(*appel des fonction de regulation de gaz*)
REGULATION_GAZ_L1(
	RESET:= MACHINE.STATE_Off,
	MANUAL:= MACHINE.STATE_Manu,
	VAC:= PRG_POMPAGE.VAC,
	DOOR := PRG_POMPAGE.DOOR,
	USER:= TRUE,
	PRM_Pos_Vanne:= ,
	PRM_Pressure:= ,
	PRM_Pressure_H:= ,
	PRM_Pressure_L:= ,
	PRM_Tim_Stab:= ,
 	PRM_Tim_Max_Stab:= REGULATION_GAZ_L1.PRM_Tim_Stab + T#30s,
	I_Pompage_Proc_Ok:= PRG_POMPAGE.POMPAGE.OP_Pompage_Proc.OK,
	I_Pompage_Sec_Ok:= PRG_POMPAGE.POMPAGE.OP_Pompage_Sec.EC
						OR PRG_POMPAGE.POMPAGE.OP_Pompage_Sec.OK, 	(*on n'attend pas la fin du pompage secondaire pour ne pas bloquer l'init*)
	I_Act_Pressure:= PRG_POMPAGE.M11.STATE_Pression,
	I_Marche_Gaz_Ok:= LIGNE_GAZ[1].OP_MARCHE.OK,
	I_Arret_Gaz_Ok:= LIGNE_GAZ[1].OP_ARRET.OK,
	I_Atm:= PRG_POMPAGE.POMPAGE.TH_Atm,
	PRM_Tim_Def_Pr:= (*config machine*),
	PRM_Tim_Ala_Pr:= (*config machine*),
	CONF_Flow_Init:= (*config machine*),
);

REGULATION_GAZ_L2(
	RESET:= MACHINE.STATE_Off,
	MANUAL:= MACHINE.STATE_Manu,
	VAC:= PRG_POMPAGE.VAC,
	DOOR := PRG_POMPAGE.DOOR,
	USER:= TRUE,
	PRM_Pos_Vanne:= ,
	PRM_Pressure:= ,
	PRM_Pressure_H:= ,
	PRM_Pressure_L:= ,
	PRM_Tim_Stab:= ,
 	PRM_Tim_Max_Stab:= REGULATION_GAZ_L2.PRM_Tim_Stab + T#30s,
	I_Pompage_Proc_Ok:= PRG_POMPAGE.POMPAGE.OP_Pompage_Proc.OK,
	I_Pompage_Sec_Ok:= PRG_POMPAGE.POMPAGE.OP_Pompage_Sec.EC
						OR PRG_POMPAGE.POMPAGE.OP_Pompage_Sec.OK, 	(*on n'attend pas la fin du pompage secondaire pour ne pas bloquer l'init*)
	I_Act_Pressure:= PRG_POMPAGE.M11.STATE_Pression,
	I_Marche_Gaz_Ok:= LIGNE_GAZ[2].OP_MARCHE.OK,
	I_Arret_Gaz_Ok:= LIGNE_GAZ[2].OP_ARRET.OK,
	I_Atm:= PRG_POMPAGE.POMPAGE.TH_Atm,
	PRM_Tim_Def_Pr:= (*config machine*),
	PRM_Tim_Ala_Pr:= (*config machine*),
	CONF_Flow_Init:= (*config machine*),
);

(*Affection des sorties*)
OUT_VG11	:=	LIGNE_GAZ[1].VGI.OUT_On;
OUT_VG12	:=	LIGNE_GAZ[2].VGI.OUT_On;
OUT_VG13	:=	LIGNE_GAZ[3].VGI.OUT_On;
OUT_VG14	:=	LIGNE_GAZ[4].VGI.OUT_On;
OUT_VGIN1	:=	VGIN[1].OUT_On;
OUT_VGIN2	:=	VGIN[2].OUT_On;
OUT_VGIN3	:=	VGIN[3].OUT_On;
OUT_VGIN4	:=	VGIN[4].OUT_On;

(*Affectation des état*)
STATE_AR :=((MACHINE.STATE_Auto OR MACHINE.STATE_Prod) AND LIGNE_GAZ[1].OP_ARRET.OK AND REGULATION_GAZ_L1.OP_ARRET.OK
			AND LIGNE_GAZ[2].OP_ARRET.OK AND REGULATION_GAZ_L2.OP_ARRET.OK AND
			LIGNE_GAZ[3].OP_ARRET.OK AND LIGNE_GAZ[4].OP_ARRET.OK) OR
			(MACHINE.STATE_Manu AND LIGNE_GAZ[1].VGI.STATE_Off AND LIGNE_GAZ[2].VGI.STATE_Off AND
			LIGNE_GAZ[3].VGI.STATE_Off AND LIGNE_GAZ[4].VGI.STATE_Off);

(*défaut entrainant l'arrêt du procédé*)
STATE_Def_IProc		:=		LIGNE_GAZ[1].VGI.DEF_Off_auto.DEF OR LIGNE_GAZ[1].VGI.DEF_On_Imposs.DEF OR LIGNE_GAZ[1].VGI.DEF_Off_Imposs.DEF OR
							LIGNE_GAZ[1].OP_MARCHE.DEF_ON_REJECTED.DEF OR LIGNE_GAZ[1].OP_ARRET.DEF_AUTO_ON.DEF OR
							LIGNE_GAZ[2].VGI.DEF_Off_auto.DEF OR LIGNE_GAZ[2].VGI.DEF_On_Imposs.DEF OR LIGNE_GAZ[2].VGI.DEF_Off_Imposs.DEF OR
							LIGNE_GAZ[2].OP_MARCHE.DEF_ON_REJECTED.DEF OR LIGNE_GAZ[2].OP_ARRET.DEF_AUTO_ON.DEF OR
							LIGNE_GAZ[3].VGI.DEF_Off_auto.DEF OR LIGNE_GAZ[3].VGI.DEF_On_Imposs.DEF OR LIGNE_GAZ[3].VGI.DEF_Off_Imposs.DEF OR
							LIGNE_GAZ[3].OP_MARCHE.DEF_ON_REJECTED.DEF OR LIGNE_GAZ[3].OP_ARRET.DEF_AUTO_ON.DEF OR
							LIGNE_GAZ[4].VGI.DEF_Off_auto.DEF OR LIGNE_GAZ[4].VGI.DEF_On_Imposs.DEF OR LIGNE_GAZ[4].VGI.DEF_Off_Imposs.DEF OR
							LIGNE_GAZ[4].OP_MARCHE.DEF_ON_REJECTED.DEF OR LIGNE_GAZ[4].OP_ARRET.DEF_AUTO_ON.DEF OR
							VGIN[1].DEF_Off_auto.DEF OR VGIN[1].DEF_Off_Imposs.DEF OR VGIN[1].DEF_On_Imposs.DEF OR
							VGIN[2].DEF_Off_auto.DEF OR VGIN[2].DEF_Off_Imposs.DEF OR VGIN[2].DEF_On_Imposs.DEF OR
							VGIN[3].DEF_Off_auto.DEF OR VGIN[3].DEF_Off_Imposs.DEF OR VGIN[3].DEF_On_Imposs.DEF OR
							VGIN[4].DEF_Off_auto.DEF OR VGIN[4].DEF_Off_Imposs.DEF OR VGIN[4].DEF_On_Imposs.DEF OR
							DG[1].DEF_SURV.DEF OR DG[2].DEF_SURV.DEF OR DG[3].DEF_SURV.DEF OR DG[4].DEF_SURV.DEF OR
							REGULATION_GAZ_L1.OP_MARCHE.DEF_ON_REJECTED.DEF OR REGULATION_GAZ_L1.OP_ARRET.DEF_AUTO_ON.DEF OR
							REGULATION_GAZ_L2.OP_MARCHE.DEF_ON_REJECTED.DEF OR REGULATION_GAZ_L2.OP_ARRET.DEF_AUTO_ON.DEF OR
							REGULATION_GAZ_L1.STATE_NOK OR REGULATION_GAZ_L2.STATE_NOK;

END_FUNCTION_BLOCK

// ---- POUs/Fonction/FONCTIONS GAZ/BLOCK_LIGNE_GAZ.TcPOU
FUNCTION_BLOCK BLOCK_LIGNE_GAZ
(* Gestion d'une ligne de gaz avec une vanne et un debitmètre *)

(****************historique des versions*****************************)

(* Version 1-0 - AB - VERSION INITIALE - base 6619, changement de classe de DG (MFC_BKH => MFC_MKS1179_AB*)
(* Version 2-0 - HG - Adaptation pour journal des évènements externe - 27/06/2011*)
(* Version 3.0 - AB - Variable IN_OUT DG_Prm_Flow dissociée en deux variabes, permettant de l'écrire hors appel à la fonction dans le PRG*)

(*************************************************************************)

VAR_INPUT
(*informations générales*)
	RESET:					BOOL;		(* Condition de réinitialisation de la fonction *)
	MANUAL:					BOOL;		(* Ordre de commmande manuel de la fonction *)
	CTRL_PLC:				BOOL;		(* Mode de contrôle de la fonction - 0 = contrôle depuis l'IHM - 1=contrôle depuis l'automate*)
(*sécurité*)
	VAC:					BOOL;		(* Entrée d'interlock de vide*)
	DOOR:					BOOL;		(* Entrée d'interlock porte*)
(*Composants*)
	VGI:					BLOCK_ACTUATOR2;				(* Vanne injection de gaz de la ligne*)

(*Paramètres*)
	PRM_Disable_Surv:		BOOL;		(* Désactivation surveillance débit externe au bloc *)
	PRM_Flow:				REAL;		(* ~ (OPC : 1 : available for OPC-clients) *)	(* Consigne de débit gaz*)
	CO_Modif:				BOOL;		(* ~ (OPC : 1 : available for OPC-clients) *)	(* Demande modification en ligne*)
(*Opérations*)
	OP_MARCHE:				BLOCK_OPERATION;		(* Opération mise en gaz ligne*)
	OP_ARRET:				BLOCK_OPERATION;		(* Opération arret gaz*)
	OP_RAMPE:				BLOCK_RAMP;			(* Opération rampe de gaz*)

(*Retour débitmètre associé*)
	IN_DG_PRM_FLOW:			REAL;
END_VAR

VAR_OUTPUT
	STATE_NOK:				BOOL;		(* ~ (OPC : 1 : available for OPC-clients) *)	(* Défaut ligne de gaz*)
	STATE_Ready:			BOOL;		(* ~ (OPC : 1 : available for OPC-clients) *)	(* Mise en gaz autorisée*)
	O_SURV_DISABLE:			BOOL;		(* I_STANDARD -- Sortie de désactivation de la surveillance du débit vers le bloc MFC associé*)

(*pilotage débitmètre associé*)
	OUT_DG_PRM_FLOW:		REAL;
END_VAR

VAR_INPUT PERSISTENT
	(*Entité*)
	IsAssembly:		BOOL;			(*entité : fonction*)
	IdXML:			STRING;			(*nom entité : identifiant pour recherche dans dico*)
	TagXML:			UINT;			(*nom entité : identifiant pour recherche dans dico*)
	IdParent:		STRING;			(*MNEMO de l'appelant*)
	MNEMO:			STRING;			(*MNEMO de l'entité*)
END_VAR

VAR_IN_OUT
	(*DG_PRM_FLOW:			REAL;											(*Variable PRM flow du massflow associé*)*)
END_VAR

VAR
	FM_CO_Modif:			R_TRIG;
	VAR_Flow:				REAL;
END_VAR

(*Début de bloc*)
PRL();
(*Opération arrêt gaz*)
ACT_STOP();
(*Opération marche gaz*)
ACT_START();
(*Fin de bloc*)
POST();

ACTION ACT_START:
(*OPERATION MARCHE GAZ*)
(*Marche gaz en continu*)

OP_MARCHE(
	CTRL_PLC:= CTRL_PLC,
	RESET:= reset,
	MANUAL:=manual ,
	RESTART_ENABLE_IF_OK:=TRUE ,
	N_STEP_OP_OK:= 3,
	N_STEP_OP_NOK:=0 );

(*appel de l'action de préparation de l'opération*)
OP_MARCHE.PRL();

(*GRAFCET*)
(* initialisation du grafcet*)
IF 		OP_MARCHE.ETAPE = 0
		THEN
				OP_MARCHE.ETAPE.0 := TRUE;
(*repositionnement sur étape 0*)
ELSIF 	MANUAL OR RESET OR OP_ARRET.ETAPE.1
		THEN
				OP_MARCHE.ETAPE := 0;
				OP_MARCHE.ETAPE.0:=TRUE;
(*étape 0-1*)
ELSIF 	OP_MARCHE.ETAPE.0 AND OP_MARCHE.MARCHE_OP
		THEN
				OP_MARCHE.ETAPE.1:=TRUE;
				OP_MARCHE.ETAPE.0:=FALSE;
(*étape 1-2*)
ELSIF	OP_MARCHE.ETAPE.1 AND OP_ARRET.ETAPE.0
		THEN
				OP_MARCHE.ETAPE.2:=TRUE;
				OP_MARCHE.ETAPE.1:=FALSE;
(*étape 2-3*)
ELSIF	OP_MARCHE.ETAPE.2 AND (VGI.STATE_On OR VAR_Flow=0)
		THEN
				OP_MARCHE.ETAPE.3:=TRUE;
				OP_MARCHE.ETAPE.2:=FALSE;
(*étape 3-2*)
ELSIF	OP_MARCHE.ETAPE.3 AND
	(OP_MARCHE.MARCHE_OP OR  (FM_CO_Modif.Q AND NOT OP_RAMPE.MARCHE.EC))
		THEN
				OP_MARCHE.ETAPE.2:=TRUE;
				OP_MARCHE.ETAPE.3:=FALSE;
END_IF;
(*cloture du traitement de l'opération*)
OP_MARCHE.POST();
END_ACTION

ACTION ACT_STOP:
(*OPERATION STOP GAZ*)

OP_ARRET(
	CTRL_PLC:= CTRL_PLC,
	RESET:= reset,
	MANUAL:=manual ,
	RESTART_ENABLE_IF_OK:=FALSE ,
	N_STEP_OP_OK:= 2,
	N_STEP_OP_NOK:=0 );

(*appel de l'action de préparation de l'opération*)
OP_ARRET.PRL();

(*GRAFCET*)
(* initialisation du grafcet*)
IF 		OP_ARRET.ETAPE = 0
		THEN
				OP_ARRET.ETAPE.0 := TRUE;
(*repositionnement sur étape 0*)
ELSIF 	MANUAL OR RESET OR OP_MARCHE.ETAPE.1
		THEN
				OP_ARRET.ETAPE := 0;
				OP_ARRET.ETAPE.0:=TRUE;
(*étape 0-1*)
ELSIF 	OP_ARRET.ETAPE.0 AND OP_ARRET.MARCHE_OP
		THEN
				OP_ARRET.ETAPE.1:=TRUE;
				OP_ARRET.ETAPE.0:=FALSE;
(*étape 1-2*)
ELSIF 	OP_ARRET.ETAPE.1 AND VGI.STATE_OFF AND OP_MARCHE.Etape.0
		THEN
				OP_ARRET.ETAPE.2:=TRUE;
				OP_ARRET.ETAPE.1:=FALSE;
END_IF;

(*cloture du traitement de l'opération*)
OP_ARRET.POST();
END_ACTION

ACTION POST:
(*Etat prêt*)
STATE_READY	:=	VAC AND DOOR;

(*Autorisations*)
OP_ARRET.ON_AUTO_INT	:=	VGI.DEF_Off_auto.DEF AND NOT Manual;
OP_ARRET.ENABLE_INT		:=	TRUE;
OP_MARCHE.ENABLE_INT	:=	STATE_Ready;

(*Gestion demandes*)
FM_CO_Modif(clk:=CO_modif);

(*Gestion rampe*)
IF	FM_CO_Modif.Q AND OP_RAMPE.MARCHE.EC THEN
	OP_RAMPE.CO_Modif_Rampe	:=	TRUE;
END_IF;
OP_RAMPE.MARCHE.RESET		:=	NOT OP_MARCHE.OK;
OP_RAMPE.MARCHE.ENABLE_INT	:=	OP_MARCHE.OK;
OP_RAMPE.MARCHE.CTRL_PLC := CTRL_PLC;
OP_RAMPE(
	IN_VALUE:=IN_DG_PRM_FLOW,
	PRM_RAMPE:=PRM_Flow);

(*Gestion vanne*)
VGI.CO_On	:= 	(OP_MARCHE.Etape.2 OR OP_MARCHE.Etape.3) AND (IN_DG_PRM_FLOW>0);
VGI(
	RESET:=Reset ,
	MANUAL:=Manual ,
	EN_On_INT:=STATE_Ready);

(*Gestion débitmètre*)
IF		OP_MARCHE.Etape.2 THEN
	OUT_DG_PRM_FLOW	:=	PRM_Flow;
ELSIF	OP_MARCHE.AR AND NOT manual THEN
	OUT_DG_PRM_FLOW	:=	0.0;
ELSIF	Manual THEN
	OUT_DG_PRM_FLOW	:=	PRM_Flow;
ELSIF	OP_RAMPE.MARCHE.EC THEN
	OUT_DG_PRM_FLOW	:=	OP_RAMPE.OUT_VALUE;
END_IF

(*Gestion défauts*)
(*alarme, défaut surveillance*)
O_SURV_DISABLE		:=	NOT VGI.STATE_On OR PRM_Disable_Surv;


(*Etat défaut*)
STATE_NOK		:=	FALSE;

(*Reset demandes*)
CO_Modif	:=	FALSE;
END_ACTION

ACTION PRL:
	OP_MARCHE.IdXML		:=	'0';
	OP_MARCHE.TagXML	:=	1;

	OP_ARRET.IdXML		:=	'0';
	OP_ARRET.TagXML		:=	2;

	OP_RAMPE.IdXML		:=	'18';
	OP_RAMPE.TagXML		:=	1;

	VGI.IdXML					:=	'1';
	VGI.TagXML					:=	1;
	VGI.DEF_Off_auto.IdXML		:=	'3';
	VGI.DEF_Off_auto.TagXML		:=	11;
	VGI.DEF_Off_Imposs.IdXML	:=	'3';
	VGI.DEF_Off_Imposs.TagXML	:=	9;
	VGI.DEF_On_Imposs.IdXML		:=	'3';
	VGI.DEF_On_Imposs.TagXML	:=	6;
END_ACTION

END_FUNCTION_BLOCK

// ---- POUs/FONCTION DE BASE/BLOCK_RAMP.TcPOU
FUNCTION_BLOCK BLOCK_RAMP
(* Gestion d'une rampe *)

(****************historique des versions*****************************)

(* Version 1-0 - HG - VERSION INIITIALE*)
(* Version 2-0 - HG - Adaptation pour journal des évènements externe - 27/06/2011*)

(*************************************************************************)
VAR_INPUT
	IN_Value:						REAL;				(* Retour consigne analogique appliquée*)
	PRM_Rampe:						REAL;				(* Consigne analogique en fin de rampe*)
	PRM_Temps:						TIME;				(* Consigne de temps de rampe*)
	CO_Modif_Rampe:					BOOL;				(* Demande modification rampe en cours*)
	CO_Rampe_Suivante:				BOOL;				(* Demande arrêt segment en cours pour passage au suivant*)
	CO_Pause:						BOOL;				(* Mise en pause de la rampe tant que la demande est valide*)
	MARCHE:						BLOCK_OPERATION;		(* Opération de gestion de la rampe*)
END_VAR

VAR_OUTPUT
	OUT_Tps_ecoule:					TIME;				(* Temps de rampe écoulé*)
	OUT_Value:						REAL;				(* Consigne analogique demandée pendant la rampe*)
	STATE_Pause:					BOOL;				(* Rampe en pause*)
END_VAR

VAR_INPUT PERSISTENT
	(*Entité*)
	IsFunction:		BOOL;			(*entité : fonction*)
	IdXML:			STRING;			(*nom entité : identifiant pour recherche dans dico*)
	TagXML:			UINT;			(*nom entité : identifiant pour recherche dans dico*)
	IdParent:		STRING;			(*MNEMO de l'appelant*)
	MNEMO:			STRING;			(*MNEMO de l'entité*)
END_VAR

VAR
	TIMER_Rampe:				TON;
	VAR_Dep_Rampe:				REAL;				(* mémoire consigne départ rampe - Gestion rampe *)
	VAR_Fin_Rampe:				REAL;				(* mémoire consigne fin rampe - Gestion rampe *)
	VAR_Tps_Rampe:				TIME;				(* mémoire consigne temps de rampe - Gestion rampe *)
	FM_Modif_rampe:				R_TRIG;
	FM_Rampe_suivante:			R_TRIG;
	FM_Pause:					R_TRIG;
END_VAR

MARCHE.IdParent			:=	MNEMO;
MARCHE.MNEMO			:=	CONCAT(MNEMO,'_MARCHE');
MARCHE.IdXML			:=	'0';
MARCHE.TagXML			:=	3;

FM_Modif_rampe(clk:=CO_Modif_Rampe);
FM_Rampe_suivante(clk:=CO_Rampe_Suivante);
FM_Pause(clk:=MARCHE.Etape.6);

(*----------G7----------*)
MARCHE(
	RESTART_ENABLE_IF_OK:=TRUE ,
	N_STEP_OP_OK:=3 ,
	N_STEP_OP_NOK:=0 );

(*appel de l'action de préparation de l'opération*)
Marche.PRL();

(*GRAFCET*)
(* initialisation du grafcet*)
IF 		MARCHE.ETAPE = 0
		THEN
				MARCHE.ETAPE.0 := TRUE;
(*repositionnement sur étape 0*)
ELSIF 	MARCHE.RESET
		THEN
				MARCHE.ETAPE := 0;
				MARCHE.ETAPE.0:=TRUE;
(*étape 0-1*)
ELSIF 	MARCHE.ETAPE.0 AND MARCHE.MARCHE_OP
		THEN
				MARCHE.ETAPE.1:=TRUE;
				MARCHE.ETAPE.0:=FALSE;
(*étape 1-2*)
ELSIF	MARCHE.ETAPE.1
		THEN
				MARCHE.ETAPE.2:=TRUE;
				MARCHE.ETAPE.1:=FALSE;
(*étape 2-7*)
ELSIF	MARCHE.ETAPE.2 AND (TIMER_rampe.Q OR VAR_tps_rampe = t#0s)
		THEN
				MARCHE.ETAPE.7:=TRUE;
				MARCHE.ETAPE.2:=FALSE;
(*étape 7-3*)
ELSIF	MARCHE.ETAPE.7
		THEN
				MARCHE.ETAPE.3:=TRUE;
				MARCHE.ETAPE.7:=FALSE;
(*étape 3-4*)
ELSIF	MARCHE.ETAPE.3 AND MARCHE.MARCHE_OP
		THEN
				MARCHE.ETAPE.4:=TRUE;
				MARCHE.ETAPE.3:=FALSE;
(*étape 4-2*)
ELSIF	MARCHE.ETAPE.4
		THEN
				MARCHE.ETAPE.2:=TRUE;
				MARCHE.ETAPE.4:=FALSE;
(*étape 2-5*)
ELSIF	MARCHE.ETAPE.2 AND FM_modif_rampe.Q
		THEN
				MARCHE.ETAPE.5:=TRUE;
				MARCHE.ETAPE.2:=FALSE;
(*étape 5-2*)
ELSIF	MARCHE.ETAPE.5
		THEN
				MARCHE.ETAPE.2:=TRUE;
				MARCHE.ETAPE.5:=FALSE;
(*étape 2-4*)
ELSIF	MARCHE.ETAPE.2 AND FM_Rampe_suivante.Q
		THEN
				MARCHE.ETAPE.4:=TRUE;
				MARCHE.ETAPE.2:=FALSE;
(*étape 2-6*)
ELSIF	MARCHE.ETAPE.2 AND CO_Pause
		THEN
				MARCHE.ETAPE.6:=TRUE;
				MARCHE.ETAPE.2:=FALSE;
(*étape 6-2*)
ELSIF	MARCHE.ETAPE.6 AND NOT CO_Pause
		THEN
				MARCHE.ETAPE.2:=TRUE;
				MARCHE.ETAPE.6:=FALSE;
END_IF;

(*Cloture du traitement de l'opération*)
MARCHE.POST();

(*Mémorisation*)
IF 		MARCHE.ETAPE.1 OR MARCHE.ETAPE.4 THEN
	VAR_dep_rampe		:=	IN_VALUE;
	VAR_fin_rampe		:=	PRM_rampe;
	VAR_tps_rampe		:=	PRM_temps;
	OUT_Tps_ecoule		:=	T#0s;
ELSIF		MARCHE.ETAPE.2 THEN
	OUT_Tps_ecoule		:=	Timer_rampe.ET;
ELSIF		MARCHE.ETAPE.5 THEN
	IF PRM_temps > OUT_tps_ecoule THEN
		VAR_tps_rampe		:=	PRM_temps - OUT_tps_ecoule;
	ELSE
		VAR_tps_rampe		:=	T#0s;
	END_IF;
	VAR_dep_rampe		:=	OUT_value;
	VAR_fin_rampe		:=	PRM_rampe;
END_IF;

IF			FM_pause.Q THEN
	VAR_dep_rampe		:=	OUT_value;
	VAR_tps_rampe		:=	VAR_tps_rampe - OUT_tps_ecoule;
END_IF;

(*Temporisation*)
IF		marche.ETAPE.1 OR marche.ETAPE.4 OR marche.ETAPE.5 OR marche.Etape.6 THEN
	Timer_rampe.PT	:=	VAR_tps_rampe;
END_IF;
timer_rampe.IN	:= marche.ETAPE.2;
Timer_Rampe();

(*Sortie*)
IF 		marche.ETAPE.3 THEN
	OUT_value	:=	var_fin_rampe;
ELSIF	marche.ETAPE.2 AND (var_tps_rampe <> t#0S) THEN
		OUT_value	:= 	(VAR_fin_rampe - VAR_dep_rampe) * (TIME_TO_REAL(OUT_tps_ecoule)/TIME_TO_REAL(VAR_tps_rampe)) +VAR_dep_rampe;
ELSIF	marche.ETAPE.1 THEN
	OUT_value 	:=	IN_value;
ELSIF	MARCHE.Etape.7 THEN
	OUT_Value := VAR_fin_Rampe;
END_IF;

(*Etat*)
STATE_Pause	:=	MARCHE.Etape.6;

CO_Modif_rampe		:=	FALSE;
CO_Rampe_Suivante	:=	FALSE;
CO_Pause			:=	FALSE;

END_FUNCTION_BLOCK

// ---- POUs/Composant/GAZ/BLOCK_MFC_MKS_NoCoE.TcPOU
FUNCTION_BLOCK BLOCK_MFC_MKS_NoCoE
(* Gestion débitmètre massique MKS sur Ethercat*)

(*Copie conforme du BLOCK_MFC_BROOKS_NoCoE*)

(****************historique des versions*****************************)

(* Version 1-0 - AB - VERSION INITIALE*)
(* Version simpliste sans programmation du CoE (débitmètre bien configuré en arrivant)*)
(* Le changement de type de gaz se fait encore via la configuration machine *)
(* Pas de gestion des erreurs / alarmes internes ==> TODO? *)

(*************************************************************************)

VAR_INPUT
	I_PARAM_SYSTEM_OK:		BOOL;		(*paramétrage système ok*)
(*informations générales*)
	RESET:					BOOL;		(* Condition de réinitialisation de la fonction *)
	PRM_Flow:				REAL;		(* Consigne débit gaz*)

	(*DEF_MFC:				PRCDEF;	(* Défaut interne débitmètre*)*)
	DEF_SURV:				PRCDEF;	(* Défaut surveillance débit*)
	ALM_SURV:				PRCDEF;	(* Alarme surveillance débit*)
	VAR_DEF_SURV:			SURVPRC;	(* Condition defaut surveillance débit*)
	VAR_ALM_SURV:			SURVPRC;	(* Condition alarme surveillance débit*)

	I_SURV_DISABLE:			BOOL;		(* I_STANDARD -- option de desactivation de la surveillance du débit venant du bloc ligne de gaz*)
END_VAR

VAR_OUTPUT
	STATE_Flow:				REAL;		(* Débit gaz appliqué*)
	CONF_Util_Max_Flow:		REAL:=1;		(* Débit max gaz utilisé*)
	(*STATE_Com:				BOOL;		(* Etat communication profibus*)*)
	STATE_NOK:				BOOL;		(* Débitmètre en défaut*)
END_VAR

VAR_INPUT PERSISTENT
(*Configuration*)
	CONF_Nom_Max_Flow:		REAL:=1;		(* Débit max gaz nominal débitmètre*)
	CONF_Nom_Coef:			REAL:=1;		(* Coefficient gaz nominal débitmètre*)
	CONF_Util_Coef:			REAL:=1;		(* Coefficient gaz utilisé*)
	CONF_Nom_Name:			STRING;		(*Nom du gaz nominal*)
	CONF_Util_Name:			STRING;		(*Nom du gaz utilisé*)

	(*Entité*)
	IsComponent:		BOOL;			(*entité : composant*)
	IdXML:				STRING;			(*nom entité : identifiant pour recherche dans dico*)
	TagXML:				UINT;			(*nom entité : identifiant pour recherche dans dico*)
	IdParent:			STRING;			(*MNEMO de l'appelant*)
	MNEMO:				STRING;			(*MNEMO de l'entité*)
END_VAR

VAR
	IN_Measure		AT%I*:	REAL;
	OUT_Setpoint	AT%Q*:	REAL;

	VAR_Ret_flow:			REAL;
	VAR_Cons_flow:			REAL;
END_VAR

IdXML					:=	'7';
TagXML					:=	1;

DEF_SURV.IdXML		:=	'0';
DEF_SURV.TagXML		:=	7;

ALM_SURV.IdXml			:=	'0';
ALM_SURV.TagXml		:=	8;
ALM_SURV.Groupe		:=	1;

(*Débit max utile*)
IF CONF_Nom_Coef > 0.0 THEN
	CONF_Util_Max_Flow	:=	CONF_Nom_Max_Flow * CONF_Util_Coef / CONF_Nom_Coef;
ELSE
	CONF_Util_Max_Flow	:=	0.0;
END_IF;

(*Retour débit*)
IF CONF_Nom_Coef > 0.0 THEN
	VAR_Ret_Flow	:=	IN_Measure;		(*retour directement en réel*)
	STATE_Flow		:=	VAR_Ret_Flow * CONF_Util_Coef / CONF_Nom_Coef;
ELSE
	STATE_Flow		:=	0.0;
END_IF

(*Consigne débit*)
IF NOT reset AND PRM_Flow>0.0 AND CONF_Util_Coef > 0.0 THEN
	VAR_Cons_Flow	:=	PRM_Flow * CONF_Nom_Coef / CONF_Util_Coef;
ELSE
	VAR_Cons_Flow	:=	0.0;
END_IF;

OUT_Setpoint	:=	VAR_Cons_flow;

(*Retour état*)
STATE_NOK		:=	ALM_SURV.DEF OR DEF_SURV.DEF;

(*desactivation de la surveillance*)
ALM_SURV.DISABLE	:=	I_SURV_DISABLE;
DEF_SURV.DISABLE	:=	I_SURV_DISABLE;

(*Défaut surveillance*)
VAR_ALM_SURV(MEASURE:=STATE_Flow , SETPOINT:= PRM_Flow);
ALM_SURV.CONDITION	:=	VAR_ALM_SURV.CONDITION AND (ALM_SURV.DELAY > T#0ms) ;
ALM_SURV();

VAR_DEF_SURV(MEASURE:=STATE_Flow , SETPOINT:= PRM_Flow);
DEF_SURV.CONDITION	:=	VAR_DEF_SURV.CONDITION AND (DEF_SURV.DELAY > T#0ms) ;
DEF_SURV();

END_FUNCTION_BLOCK

// ---- POUs/FONCTION DE BASE/SURVPRC.TcPOU
FUNCTION_BLOCK SURVPRC

(* Fonction standard AC de gestion surveillance de défaut *)

(****************historique des versions*****************************)

(* Version 1-0 - HG - VERSION INIITIALE*)

(*************************************************************************)

VAR_INPUT
	MEASURE:			REAL;	(* Retour valeurs à surveillées*)
	SETPOINT:			REAL;	(* Consigne valeurs à surveillées*)

END_VAR

VAR_OUTPUT
	CONDITION:			BOOL;	(* Condition de défaut *)
END_VAR
VAR_INPUT PERSISTENT
	OFFSET:			REAL;	 (* Ecart toléré*)
END_VAR

(*Surveillance inhibée si offset = 0*)
IF OFFSET <> 0
	AND (ABS(MEASURE - SETPOINT) > OFFSET) THEN
	CONDITION := TRUE;
ELSE
	CONDITION := FALSE;
END_IF;

END_FUNCTION_BLOCK

// ---- POUs/Fonction/FONCTIONS GAZ/BLOCK_REGUL_PR_GAZ.TcPOU
FUNCTION_BLOCK BLOCK_REGUL_PR_GAZ
(* Gestion d'une fonction de régulation de la pression d'une enceinte directement sur débit de gaz
Interfaçage avec fonction de pompage avec vanne asservie
Interfaçage avec une seule ligne de gaz
Introduction du BLOCK_CONTROL_GAZ gérant le PID
*)

(****************historique des versions*****************************)

(* Version 1-0 - AB - VERSION INITIALE - aff 8415 CT200 n8 Nivarox*)

(*************************************************************************)

VAR_INPUT

(*informations générales*)
	RESET:					BOOL;		(* Condition de réinitialisation de la fonction *)
	MANUAL:					BOOL;		(* Ordre de commmande manuel de la fonction *)
	CTRL_PLC:				BOOL;		(* Mode de contrôle de la fonction - 0 = contrôle depuis l'IHM - 1=contrôle depuis l'automate*)
(*sécurité*)
	VAC:					BOOL;		(* Entrée d'interlock de vide*)
	DOOR:					BOOL;		(* Entrée d'interlock porte*)
	USER:					BOOL;		(* Entrée d'interlock utilisateur*)
(*Composants*)
	CONTROLEUR_GAZ:			BLOCK_CONTROL_GAZ;

(*Paramètres*)
	PRM_Pos_Vanne:			REAL;		(*Position fixe de la vanne secondaire*)
	PRM_Pressure:			REAL;		(*Consigne de pression à obtenir en régulation*)
	PRM_Pressure_H:			REAL;		(*Limite haute de l'intervalle de pression considéré pour regul ok*)
	PRM_Pressure_L:			REAL;		(*Limite basse de l'intervalle de pression considéré pour regul ok*)
	PRM_Tim_Stab:			TIME;		(*Temps considéré pour valider la stabilisation*)
	PRM_Tim_Max_Stab:		TIME;		(*Temps max pour obtention stabilisation, avant déclenchement défaut : doit être supérieur à PRM_tim_stab*)

	CO_Modif:				BOOL;		(* ~ (OPC : 1 : available for OPC-clients) *)	(* Demande modification en ligne*)

(*Interfaçage avec autres fonctionnalités*)
	I_Pompage_Proc_Ok:		BOOL;		(*Retour mise en position vanne asservie ok*)
	I_Pompage_Sec_Ok:		BOOL;		(*Retour pompage secondaire ok*)
	I_Act_Pressure:			REAL;		(*Retour mesure pression*)
	I_Atm:					BOOL;		(*retour d'info de chambre à H, sert à éviter de lancer le pompage sec en arrêt lors d'un init chambre ouverte*)

	I_Marche_Gaz_Ok:		BOOL;		(*Retour mise en gaz ok*)
	I_Arret_Gaz_Ok:			BOOL;		(*Retour arret gaz ok*)
	VAR_Controleur_Gaz_Ok:	BOOL;		(*Retour mise en marche controleur gaz ok*)

(*Opérations*)
	OP_MARCHE:				BLOCK_OPERATION;		(* Opération mise en gaz ligne*)
	OP_ARRET:				BLOCK_OPERATION;		(* Opération arret gaz*)

(*Défaut*)
	DEF_Pression:				PRCDEF;			(*Défaut d'obtention de la pression*)
	DEF_Surv_Pression:			PRCDEF;			(*Défaut de surveillance de la pression - perte du critère de stabilisation*)
	ALA_Surv_Pression:			PRCDEF;			(*Alarme de surveillance de la rpession - perte du critère de stabilisation*)
END_VAR

VAR_OUTPUT
	(*gestion fonctions externes*)
	RQ_Ctrl_Pompage:			BOOL;		(*Prise en charge pompage*)
	RQ_Ctrl_Gaz:				BOOL;		(*Prise en charge gaz*)

	(*demandes pour fonctions externes*)
	RQ_Pompage_Proc:		BOOL;		(*mise en laminage*)
	RQ_Pompage_Sec:			BOOL;		(*pompage secondaire*)
	RQ_Marche_Gaz:			BOOL;		(*mise en gaz*)
	RQ_Arret_Gaz:			BOOL;		(*arret gaz*)

	STATE_Ready:			BOOL;		(* Etat prêt*)
	STATE_NOK:				BOOL;		(* Défaut asservissement pression*)
END_VAR

VAR_INPUT PERSISTENT
	PRM_Tim_Def_Pr:			TIME;
	PRM_Tim_Ala_Pr:			TIME;
	CONF_Flow_Init:			REAL;		(*consigne de gaz initiale*)

	(*Entité*)
	IsAssembly:		BOOL;			(*entité : fonction*)
	IdXML:			STRING;			(*nom entité : identifiant pour recherche dans dico*)
	TagXML:			UINT;			(*nom entité : identifiant pour recherche dans dico*)
END_VAR

VAR
	VAR_Start_Controleur_Gaz_Ok:	BOOL;		(*Mise en marche controleur gaz ok*)
	VAR_Stop_Controleur_Gaz_Ok:		BOOL;		(*Arret controleur gaz ok*)
	VAR_Stab_Pression_Ok:			BOOL;		(*Stabilisation pression ok*)

	VAR_Attente_Stab:				BOOL;		(*falg indiquant que l'on est dans l'étape d'attente de stabilsiation de la pression*)
	 VAR_Surv_Pression:				BOOL;		(*flag de demande de surveillance de maintien de la pression stabilisée*)

	FM_CO_Modif:			R_TRIG;

	(*fronts montants*)
	FM_Arret_2:				R_TRIG;
	FM_Arret_4:				R_TRIG;
	FM_Marche_4:			R_TRIG;
	FM_Marche_6:			R_TRIG;

	(*timer*)
	TIMER_Valid_Press_Ok:	TON;

	TIMER_Marche2:			TON;
	TIMER_Arret5:			TON;

END_VAR

(*Début de bloc*)
PRL();
(*Opération arrêt gaz*)
ACT_STOP();
(*Opération marche gaz*)
ACT_START();
(*Fin de bloc*)
POST();

ACTION ACT_START:
(*OPERATION MARCHE GAZ*)
(*Marche gaz en continu*)

OP_MARCHE(
	CTRL_PLC:= CTRL_PLC,
	RESET:= reset,
	MANUAL:=manual ,
	RESTART_ENABLE_IF_OK:=TRUE ,
	N_STEP_OP_OK:= 12,
	N_STEP_OP_NOK:=0 );

(*appel de l'action de préparation de l'opération*)
OP_MARCHE.PRL();

(*GRAFCET*)
(* initialisation du grafcet*)
IF 		OP_MARCHE.ETAPE = 0
		THEN
				OP_MARCHE.ETAPE.0 := TRUE;
(*repositionnement sur étape 0*)
ELSIF 	MANUAL OR RESET OR OP_ARRET.ETAPE.1
		THEN
				OP_MARCHE.ETAPE := 0;
				OP_MARCHE.ETAPE.0:=TRUE;
(*étape 0-1*)
ELSIF 	OP_MARCHE.ETAPE.0
		AND OP_MARCHE.MARCHE_OP
		THEN
				OP_MARCHE.ETAPE.1:=TRUE;
				OP_MARCHE.ETAPE.0:=FALSE;
(*étape 1-2*)
ELSIF	OP_MARCHE.ETAPE.1
		AND OP_ARRET.ETAPE.0
		THEN
				OP_MARCHE.ETAPE.2:=TRUE;
				OP_MARCHE.ETAPE.1:=FALSE;
(*étape 2-3 ==> prise de controle pompage et gaz*)
ELSIF	OP_MARCHE.ETAPE.2
		AND Timer_Marche2.Q
		THEN
				OP_MARCHE.ETAPE.3:=TRUE;
				OP_MARCHE.ETAPE.2:=FALSE;
(*étape 3-4*)
ELSIF	OP_MARCHE.ETAPE.3
		THEN
				OP_MARCHE.ETAPE.4:=TRUE;
				OP_MARCHE.ETAPE.3:=FALSE;
(*étape 4-5 ==> mise en pompage procédé*)
ELSIF	OP_MARCHE.ETAPE.4
		AND I_Pompage_Proc_Ok
		THEN
				OP_MARCHE.ETAPE.5:=TRUE;
				OP_MARCHE.ETAPE.4:=FALSE;
(*étape 5-6*)
ELSIF	OP_MARCHE.ETAPE.5
		THEN
				OP_MARCHE.ETAPE.6:=TRUE;
				OP_MARCHE.ETAPE.5:=FALSE;
(*étape 6-7 ==> mise en marche gaz*)
ELSIF	OP_MARCHE.ETAPE.6
		AND I_Marche_Gaz_Ok
		THEN
				OP_MARCHE.ETAPE.7:=TRUE;
				OP_MARCHE.ETAPE.6:=FALSE;
(*étape 7-8*)
ELSIF	OP_MARCHE.ETAPE.7
		THEN
				OP_MARCHE.ETAPE.8:=TRUE;
				OP_MARCHE.ETAPE.7:=FALSE;
(*étape 8-9 ==> marche controlleur gaz*)
ELSIF	OP_MARCHE.ETAPE.8
		(*AND VAR_Start_Controleur_Gaz_Ok*)
		THEN
				OP_MARCHE.ETAPE.9:=TRUE;
				OP_MARCHE.ETAPE.8:=FALSE;
(*étape 9-10*)
ELSIF	OP_MARCHE.ETAPE.9
		THEN
				OP_MARCHE.ETAPE.10:=TRUE;
				OP_MARCHE.ETAPE.9:=FALSE;
(*étape 10-11*)
ELSIF	OP_MARCHE.ETAPE.10
		AND VAR_Stab_Pression_ok
		THEN
				OP_MARCHE.ETAPE.11:=TRUE;
				OP_MARCHE.ETAPE.10:=FALSE;
(*étape 11-12*)
ELSIF	OP_MARCHE.ETAPE.11
		THEN
				OP_MARCHE.ETAPE.12:=TRUE;
				OP_MARCHE.ETAPE.11:=FALSE;

(*étape 12-1*)
ELSIF	OP_MARCHE.Etape.12
		AND OP_MARCHE.MARCHE_OP
		THEN
				OP_MARCHE.Etape.1 := TRUE;
				OP_MARCHE.Etape.12 := FALSE;
END_IF;
(*cloture du traitement de l'opération*)
OP_MARCHE.POST();
END_ACTION

ACTION ACT_STOP:
(*OPERATION STOP GAZ*)

OP_ARRET(
	CTRL_PLC:= CTRL_PLC,
	RESET:= reset,
	MANUAL:=manual ,
	ON_AUTO_INT:=	CONTROLEUR_GAZ.STATE_Nok
					OR DEF_Pression.DEF
					OR DEF_Surv_Pression.DEF,
	RESTART_ENABLE_IF_OK:=TRUE ,
	N_STEP_OP_OK:= 6,
	N_STEP_OP_NOK:=0 );

(*appel de l'action de préparation de l'opération*)
OP_ARRET.PRL();

(*GRAFCET*)
(* initialisation du grafcet*)
IF 		OP_ARRET.ETAPE = 0
		THEN
				OP_ARRET.ETAPE.0 := TRUE;
(*repositionnement sur étape 0*)
ELSIF 	MANUAL OR RESET OR OP_MARCHE.ETAPE.1
		THEN
				OP_ARRET.ETAPE := 0;
				OP_ARRET.ETAPE.0:=TRUE;
(*étape 0-1*)
ELSIF 	OP_ARRET.ETAPE.0
		AND OP_ARRET.MARCHE_OP
		THEN
				OP_ARRET.ETAPE.1:=TRUE;
				OP_ARRET.ETAPE.0:=FALSE;
(*étape 1-2*)
ELSIF 	OP_ARRET.ETAPE.1
		AND OP_MARCHE.Etape.0
		THEN
				OP_ARRET.ETAPE.2:=TRUE;
				OP_ARRET.ETAPE.1:=FALSE;
(*étape 2-3 ==> arrêt controlleur gaz et arrêt ligne gaz*)
ELSIF 	OP_ARRET.ETAPE.2
		(*AND VAR_Stop_Controleur_Gaz_Ok*)
		AND I_Arret_Gaz_Ok
		THEN
				OP_ARRET.ETAPE.3:=TRUE;
				OP_ARRET.ETAPE.2:=FALSE;
(*étape 3-4*)
ELSIF 	OP_ARRET.ETAPE.3
		THEN
				OP_ARRET.ETAPE.4:=TRUE;
				OP_ARRET.ETAPE.3:=FALSE;
(*étape 4-5*)
ELSIF 	OP_ARRET.ETAPE.4
		AND (I_Pompage_Sec_Ok OR I_Atm)
		THEN
				OP_ARRET.ETAPE.5:=TRUE;
				OP_ARRET.ETAPE.4:=FALSE;
(*étape 5-6*)
ELSIF 	OP_ARRET.ETAPE.5
		AND TIMER_Arret5.Q
		THEN
				OP_ARRET.ETAPE.6:=TRUE;
				OP_ARRET.ETAPE.5:=FALSE;
(*étape 6-1*)
ELSIF	OP_ARRET.Etape.6
		AND OP_ARRET.MARCHE_OP
		THEN
				OP_ARRET.Etape.1 := TRUE;
				OP_ARRET.Etape.6 := FALSE;

END_IF;

(*cloture du traitement de l'opération*)
OP_ARRET.POST();
END_ACTION

ACTION POST:
(*Etat prêt*)
STATE_READY	:=	VAC AND DOOR AND USER;

(*Autorisations*)
OP_ARRET.ENABLE_INT		:=	TRUE;
OP_MARCHE.ENABLE_INT	:=	STATE_Ready;

(*timers*)
TIMER_Marche2.IN := OP_MARCHE.Etape.2;
TIMER_Marche2.PT := T#100ms;
TIMER_Marche2();

TIMER_Arret5.IN := OP_ARRET.Etape.5;
TIMER_Arret5.PT := T#100ms;
TIMER_Arret5();

(*Gestion mode de controle des fonctions externes*)
IF		OP_MARCHE.Etape.2 THEN
			RQ_Ctrl_Pompage	:=	TRUE;
			RQ_Ctrl_Gaz			:=	TRUE;
ELSIF	OP_ARRET.Etape.5
		OR MANUAL
		OR RESET
		THEN
			RQ_Ctrl_Pompage	:=	FALSE;
			RQ_Ctrl_Gaz			:=	FALSE;
END_IF

(*Gestion controleur gaz*)
CONTROLEUR_GAZ.PRM_Pressure		:=	PRM_Pressure;
CONTROLEUR_GAZ.I_Act_Pressure		:=	I_Act_Pressure;

IF OP_MARCHE.Etape.8 THEN
	CONTROLEUR_GAZ.CO_On	:=	TRUE;
ELSIF OP_ARRET.Etape.2
		OR MANUAL
		OR RESET THEN
	CONTROLEUR_GAZ.CO_On	:=	FALSE;
END_IF

CONTROLEUR_GAZ(
		RESET	:=	RESET,
					);

(*Gestion variables internes*)
(*attente stabilisation pression*)
IF op_marche.Etape.10 THEN
	VAR_Attente_Stab		:=	TRUE;
ELSE
	VAR_Attente_Stab		:=	FALSE;
END_IF

(*stabilisation pression ok*)
TIMER_Valid_Press_OK.IN		:=		(
								(
								(I_Act_Pressure >= PRM_Pressure_L)
								AND (I_Act_Pressure <= PRM_Pressure_H)
								) OR (PRM_Tim_Stab = T#0ms)
									)
								(*AND NOT VAR_Prm_Pression_modifie ;*);
TIMER_Valid_Press_OK.PT		:=	PRM_Tim_Stab;
TIMER_Valid_Press_OK();
VAR_Stab_Pression_Ok			:=	TIMER_Valid_Press_ok.Q;

(*surveillance pression*)
IF OP_MARCHE.Etape.11 OR OP_MARCHE.Etape.12 THEN
	VAR_Surv_Pression	:=	TRUE;
ELSE
	VAR_Surv_Pression	:=	FALSE;
END_IF


(*Prise en charge des fonctions externes - passage des consignes*)
RQ_Arret_Gaz		:=	FM_Arret_2.Q;
RQ_Pompage_Sec	:=	FM_Arret_4.Q AND NOT I_Atm;
RQ_Pompage_Proc	:=	FM_Marche_4.Q;
RQ_Marche_Gaz		:=	FM_Marche_6.Q;


(*Gestion défauts*)
DEF_Pression.Condition	:= 	NOT VAR_Stab_Pression_Ok
							AND VAR_Attente_Stab
							AND NOT MANUAL
							AND NOT RESET
							AND (PRM_Tim_Max_Stab > T#0ms);
DEF_Pression(DELAY		:=	PRM_Tim_Max_Stab);

(*défaut de surveillance de la pression - l'état STATE_Press_Ok est perdu pendant un temps supérieur à PRM_TIM_SURV_PR *)
DEF_Surv_Pression.CONDITION	:=	NOT VAR_Stab_Pression_Ok
									AND VAR_Surv_Pression
									AND NOT MANUAL
									AND NOT RESET;
DEF_Surv_Pression(DELAY:=PRM_Tim_Def_Pr);


(*alarme de surveillance de la pression - l'état STATE_Press_Ok est perdu pendant un temps supérieur à PRM_ALA_SURV_PR*)
ALA_Surv_Pression.CONDITION 	:=	NOT VAR_Stab_Pression_Ok
									AND VAR_Surv_Pression
									AND NOT MANUAL
									AND NOT RESET;
ALA_Surv_Pression(DELAY:=PRM_Tim_Ala_Pr);


(*Etat défaut*)
STATE_NOK		:=	DEF_Pression.DEF OR DEF_Surv_Pression.DEF OR CONTROLEUR_GAZ.STATE_Nok;

(*Reset demandes*)
CO_Modif	:=	FALSE;
END_ACTION

ACTION PRL:
	OP_MARCHE.IdXML		:=	'0';
	OP_MARCHE.TagXML	:=	1;

	OP_ARRET.IdXML		:=	'0';
	OP_ARRET.TagXML		:=	2;

	DEF_Pression.IdXml				:=	'16';
	DEF_Pression.TagXml				:=	8;

	DEF_Surv_Pression.IdXml			:=	'16';
	DEF_Surv_Pression.TagXml		:=	11;

	ALA_Surv_Pression.IdXml			:=	'16';
	ALA_Surv_Pression.TagXml		:=	10;
	ALA_Surv_Pression.Groupe		:=	1;


(*fronts montants*)
FM_Arret_2(clk := OP_ARRET.Etape.2);
FM_Arret_4(clk := OP_ARRET.Etape.4);
FM_Marche_4(clk := OP_MARCHE.Etape.4);
FM_Marche_6(clk := OP_MARCHE.Etape.6);
END_ACTION

END_FUNCTION_BLOCK

// ---- POUs/Composant/GAZ/BLOCK_CONTROL_GAZ.TcPOU
FUNCTION_BLOCK BLOCK_CONTROL_GAZ
(* Gestion d'un controleur de débit de gaz interne Bechkoff pour régulation de pression par débit de gaz*)

(****************historique des versions*****************************)

(* Version 1-0 - AB - VERSION INITIALE - aff 8415 : CT200 n8 Nivarox*)

(*************************************************************************)

VAR_INPUT
(*informations générales*)
	RESET:					BOOL;		(* Condition de réinitialisation du controlleur*)

	(*Marche régulation*)
	CO_On:					BOOL;		(*demande de marche du PID*)

	(*Consignes*)
	PRM_Pressure:			REAL;		(* Consigne de pression*)

	(*retours d'informations*)
	I_Act_Pressure:			REAL;		(*Feedback pressure*)

	(*Défauts*)
	DEF_Internal:			PRCDEF;	(*Controlleur PID en défaut interne*)
END_VAR

VAR_OUTPUT
	STATE_Flow:				REAL;		(* Débit gaz appliqué*)

	STATE_Nok:				BOOL;		(*controlleur en défaut*)
END_VAR

VAR_INPUT PERSISTENT
	(*Configuration*)
	CONF_Kp:		REAL;			(*composante P*)
	CONF_Tn:		REAL;			(*Composante I (s)*)
	CONF_Tv:		REAL;			(*Composante D (s)*)
	CONF_Td:		REAL;			(*Composante damping time*)

	(*Entité*)
	IsComponent:	BOOL;			(*entité : composant*)
	IdXML:			STRING;			(*nom entité : identifiant pour recherche dans dico*)
	TagXML:			UINT;			(*nom entité : identifiant pour recherche dans dico*)
END_VAR

VAR
	VAR_Ctrl_PID:	FB_BasicPID;
END_VAR

IdXML					:=	'7';
TagXML					:=	4;

DEF_Internal.IdXML		:=	'0';
DEF_Internal.TagXML		:=	6;


(*configuratrion du PID*)
VAR_Ctrl_PID.fKp				:=	CONF_Kp;		(*P*)
VAR_Ctrl_PID.fTn				:=	CONF_Tn;		(*I*)
VAR_Ctrl_PID.fTv				:=	CONF_Tv;		(*D*)
VAR_Ctrl_PID.fTd				:=	CONF_Td;		(*damping*)
VAR_Ctrl_PID.fCtrlCycleTime		:=	1;				(*controle toutes les secondes, dans un premier temps*)


(*affectation des entrées*)
VAR_Ctrl_PID.fActualValue		:=	I_Act_Pressure;	(*feedback pression*)
VAR_Ctrl_PID.fSetpointValue		:=	PRM_Pressure;	(*consigne pression*)

(*lancement de la régulation PID sur Co_on et pas reset*)
VAR_Ctrl_PID(
		bReset 	:=	NOT CO_On OR RESET,
);

(*Défaut interne*)
DEF_Internal.CONDITION	:=	(VAR_Ctrl_PID.nErrorStatus > 0);
DEF_Internal.DELAY		:=	T#1s;
DEF_Internal();


(*retours controlleur*)
STATE_Flow		:=	LREAL_TO_REAL(VAR_Ctrl_PID.fCtrlOutput);		(*sortie du PID remise à zéro du bit reset, donc ok pour raz de state_flow*)
STATE_NOK		:=	DEF_internal.DEF;

END_FUNCTION_BLOCK

// ---- POUs/Programme/BLOCK_PRG_VERRINE.TcPOU
FUNCTION_BLOCK BLOCK_PRG_VERRINE
VAR_INPUT
	VERRINE:						BLOCK_VERRINE;
	BUZZER:							BLOCK_BUZZER;
END_VAR
VAR_OUTPUT
	(*Verrine*)
	OUT_Vert		AT%Q*:			BOOL;	(*allumage vert*)
	OUT_Rouge		AT%Q*:			BOOL;	(*allumage rouge*)
	OUT_Orange		AT%Q*:			BOOL;	(*allumage orange*)
	OUT_Buzzer		AT%Q*:			BOOL;
END_VAR
VAR
	VAR_Def_non_bloquant:	BOOL;

	VAR_Mem_MultiBip:		BOOL;
	TIMER_MultiBip:			TON;
	VAR_Mem_Buzz_Cont1:		BOOL;
	TIMER_Buzz_Cont1:		TON;
	FM_Proc_OK:				ARRAY[0..25] OF R_TRIG;		(*depend du nombre de slots de la cassette*)
	FD_Prod:				F_TRIG;						(*front descendant du state_prod*)
	VAR_I:					USINT;
END_VAR


(*Défauts non bloquants en procédé*)
VAR_def_non_bloquant	:=	PRG_GAZ.DG[1].ALM_SURV.DEF OR PRG_GAZ.DG[2].ALM_SURV.DEF
							OR PRG_GAZ.REGULATION_GAZ_L1.ALA_Surv_Pression.DEF OR PRG_GAZ.REGULATION_GAZ_L2.ALA_Surv_Pression.DEF
							OR PRG_POMPAGE.POMPAGE.VS11.ALA_Surv_Pression.DEF 
							OR PRG_POMPAGE.POMPAGE.VS11.DEF_Off.DEF OR PRG_POMPAGE.POMPAGE.VS11.DEF_On.DEF OR PRG_POMPAGE.POMPAGE.VS11.DEF_Position.DEF OR PRG_POMPAGE.POMPAGE.VS11.DEF_Pression.DEF
							OR PRG_POMPAGE.POMPAGE.VP11.DEF_Off.DEF OR PRG_POMPAGE.POMPAGE.VP11.DEF_On.DEF OR PRG_POMPAGE.POMPAGE.VP11.DEF_Sensor.DEF
							OR PRG_POMPAGE.POMPAGE.DEF_Vent.DEF 
							OR PRG_POMPAGE.POMPAGE.PR11.DEF_On.DEF
							OR PRG_EVAP.EVAPS1.DEF_QZ_CTRL_RATE.DEF OR PRG_EVAP.EVAPS2.DEF_QZ_CTRL_RATE.DEF OR PRG_EVAP.EVAPS3.DEF_QZ_CTRL_RATE.DEF
							OR PRG_EVAP.XTC3.STATE_NOK;						


(*------------------------------------------------------------------GESTION VERRINE----------------------------------------------------------------------------*)

VERRINE.RESET := MACHINE.STATE_Off;

(*Rouge fixe : MACHINE EN AUTOMATIE, PORTE FERMEE SANS PRODUCTION OU PRODUTION INTERROMPUE*)
VERRINE.I_rouge_cont	:=	MACHINE.STATE_Auto AND PRG_POMPAGE.DOOR AND (NOT MACHINE.STATE_Prod OR MACHINE.STATE_interrupted);

(*Rouge clignottant : NU*)
VERRINE.I_rouge_cligno	:=	FALSE;

(*Orange fixe : PROCEDE EN COURS ET DEFAUT NON BLOQUANT *)
VERRINE.I_orange_cont	:= 	MACHINE.STATE_Prod AND VAR_Def_non_bloquant;

(*Orange clignotant : NU*)
VERRINE.I_orange_cligno := 	FALSE;

(*Vert fixe : PROCEDE EN COURS ET PAS DE DEFAUT NON BLOQUANT*)
VERRINE.I_vert_cont 	:= 	MACHINE.STATE_Prod AND NOT VAR_Def_non_bloquant;

(*vert clignotant : NU*)
VERRINE.I_vert_cligno 	:=	FALSE;

VERRINE();

OUT_Orange  :=	VERRINE.OUT_orange;
OUT_Rouge	:=	VERRINE.OUT_rouge;
OUT_Vert	:=	VERRINE.OUT_vert;


(*------------------------------------------------------------------------------------GESTION BUZZER-----------------------------------------------------------------------*)
(*
(*gestion front montant fin procédé pour chaque plaque*)
FOR VAR_I := 0 TO 25 (*10*) DO
	FM_Proc_OK[VAR_I].CLK	:=	(K7.SUBSTRAT[VAR_I].STATE_Process = 3);
	FM_Proc_OK[VAR_I];
END_FOR
IF 	FM_Proc_OK[0].Q
	OR FM_Proc_OK[1].Q OR FM_Proc_OK[2].Q OR FM_Proc_OK[3].Q OR FM_Proc_OK[4].Q OR FM_Proc_OK[5].Q
	OR FM_Proc_OK[6].Q OR FM_Proc_OK[7].Q OR FM_Proc_OK[8].Q OR FM_Proc_OK[9].Q OR FM_Proc_OK[10].Q
	OR FM_Proc_OK[11].Q OR FM_Proc_OK[12].Q OR FM_Proc_OK[13].Q OR FM_Proc_OK[14].Q OR FM_Proc_OK[15].Q
	OR FM_Proc_OK[16].Q OR FM_Proc_OK[17].Q OR FM_Proc_OK[18].Q OR FM_Proc_OK[19].Q OR FM_Proc_OK[20].Q
	OR FM_Proc_OK[21].Q OR FM_Proc_OK[22].Q OR FM_Proc_OK[23].Q OR FM_Proc_OK[24].Q OR FM_Proc_OK[25].Q THEN
		VAR_Mem_Buzz_Cont1	:=	TRUE;
ELSIF TIMER_Buzz_Cont1.Q THEN
		VAR_Mem_Buzz_Cont1	:=	FALSE;
END_IF
*)

(*
BUZZER(
	I_DEF_Continu1:= 				TIMER_Buzz_Cont1.Q,
	I_DEF_Continu2:= 				FALSE,
	I_DEF_Alternatif:= 				FALSE,
	I_DEF_MultiBip:= 				FALSE,
	I_DEF_Permanent:= 			FALSE,
	RESET:= 					ENCEINTE_10.STATE_Off,
	PRM_Tp_Continu1:= 			T#5s,
	PRM_Tp_Continu2:= 			T#2s,
	PRM_Tp_Bip_Alternatif:= 		T#2s,
	PRM_Tp_Tempo_Alternatif:= 	T#2s,
	PRM_Tp_MultiBip1:= 			T#500ms,
	PRM_Tp_MultiBip2:= 			T#30s,
	PRM_Tp_Tempo_MultiBip:= 	T#2m,
	PRM_Alternatif_Temporise:= 	FALSE,
	PRM_MultiBip_Temporise:= 	FALSE,
	PRM_Acq_Continu1:= 			FALSE,
	PRM_Acq_Continu2:= 			FALSE,
	PRM_Acq_Alternatif:= 			FALSE,
	PRM_Acq_MultiBip:= 			TRUE,
	PRM_Acq_Permanent:= 		FALSE,
	PRM_Nb_Bip:=				2,
);
OUT_Buzzer	:=	BUZZER.OUT_Buzzer;*)

END_FUNCTION_BLOCK

// ---- POUs/Composant/BLOCK_VERRINE.TcPOU
FUNCTION_BLOCK BLOCK_VERRINE
(*Block de gestion de verrine 3 couleurs - clignotement possible pour chacune d'elles*)

(****************historique des versions*****************************)

(* Version 1-0 - AB - VERSION INITIALE*)
(* Version 2-0 - HG - Sans block PWM*)

(*************************************************************************)

VAR_INPUT

	I_vert_cont: 			BOOL := FALSE;		(*demande allumage vert continu*)
	I_vert_cligno:			BOOL := FALSE;		(*demande allumage vert clignotant*)
	I_orange_cont:			BOOL := FALSE;
	I_orange_cligno:		BOOL := FALSE;
	I_rouge_cont:			BOOL := FALSE;
	I_rouge_cligno:			BOOL := FALSE;
	RESET:					BOOL;		(*demande de reset *)

END_VAR


VAR_OUTPUT
	OUT_vert: 		BOOL;		(*allumage vert*)
	OUT_orange:		BOOL;
	OUT_rouge:		BOOL;

END_VAR


VAR
	(*variables de gestion du clignotement*)
	VAR_Alternatif_vert:				BLOCK_CLIGNOTANT_V0_0;
	VAR_Alternatif_orange:				BLOCK_CLIGNOTANT_V0_0;
	VAR_Alternatif_rouge:				BLOCK_CLIGNOTANT_V0_0;

END_VAR

(*entrées alternatives*)
VAR_Alternatif_vert.CONF_Period_Off		:=	T#1S;
VAR_Alternatif_vert.CONF_Period_Off		:=	T#1S;
VAR_Alternatif_orange.CONF_Period_Off	:=	T#1S;
VAR_Alternatif_orange.CONF_Period_Off	:=	T#1S;
VAR_Alternatif_rouge.CONF_Period_Off	:=	T#1S;
VAR_Alternatif_rouge.CONF_Period_Off	:=	T#1S;

(*vert*)
VAR_Alternatif_vert(IN_On	:=	I_vert_cligno AND NOT RESET);

(*orange*)
VAR_Alternatif_orange(IN_On	:=	I_orange_cligno AND NOT RESET);

(*rouge*)
VAR_Alternatif_rouge(IN_On	:=	I_rouge_cligno AND NOT RESET);

(*envoi des sorties*)
OUT_vert := VAR_Alternatif_vert.STATE_ON OR (I_vert_cont AND NOT RESET);
OUT_orange := VAR_Alternatif_orange.STATE_ON OR (I_orange_cont AND NOT RESET);
OUT_rouge := VAR_Alternatif_rouge.STATE_ON OR  (I_rouge_cont AND NOT RESET);

END_FUNCTION_BLOCK

// ---- POUs/FONCTION DE BASE/BLOCK_CLIGNOTANT_V0_0.TcPOU
FUNCTION_BLOCK BLOCK_CLIGNOTANT_V0_0
VAR_INPUT
	IN_On:				BOOL;			(*demande de marche*)
END_VAR

VAR_INPUT PERSISTENT
	CONF_Period_On:		TIME:= T#2S;	(*durée de maintien d'allumage*)	
	CONF_Period_Off:	TIME:= T#2S;	(*durée de l'arrêt d'allumage*)
END_VAR

VAR_OUTPUT
	STATE_ON:			BOOL;			(*allumage*)
END_VAR

VAR
	TIMER_On:			TP;
	TIMER_Off:			TP;
END_VAR

TIMER_On.PT		:=	CONF_Period_On;
TIMER_On.IN		:=	IN_On
					AND NOT TIMER_Off.Q;
TIMER_On();

TIMER_Off.PT	:=	CONF_Period_Off;
TIMER_Off.IN	:=	IN_On
					AND NOT TIMER_On.Q;
TIMER_Off();

STATE_ON		:=	TIMER_On.Q and IN_On;

END_FUNCTION_BLOCK

// ---- POUs/Composant/VERRINE/BLOCK_BUZZER.TcPOU
FUNCTION_BLOCK BLOCK_BUZZER
VAR_INPUT
	I_DEF_Continu1:				BOOL:=FALSE;		(*Déclenchement bip continu temporisé 1*)
	I_DEF_Continu2:				BOOL:=FALSE;		(*Déclenchement bip continu temporisé 2*)
	I_DEF_Alternatif:			BOOL:=FALSE;		(*Déclenchement bip alternatif*)
	I_DEF_MultiBip:				BOOL:=FALSE;		(*Déclenchement multi bip*)
	I_DEF_Permanent:			BOOL:=FALSE;		(*Déclenchement bip permanent*)
	M_ACQ:						BOOL;				(*Acquittement buzzer et inhibition*)
	RESET:						BOOL;
END_VAR

VAR_OUTPUT
	OUT_Buzzer:					BOOL;
END_VAR

VAR
	VAR_Alternatif:				BLOCK_CLIGNOTANT_V0_0;
	VAR_MultiBip:				BLOCK_CLIGNOTANT_V0_0;
	TIMER_Continu1:				TP;
	TIMER_Continu2:				TP;
	TIMER_Alternatif:			TP;
	TIMER_MultiBip:				TP;
	TIMER_MultiBip2:			TON;
	FM_Continu1:				R_TRIG;
	FM_Continu2:				R_TRIG;
	FM_Alternatif:				R_TRIG;
	FM_MultiBip:				R_TRIG;
	FM_Permanent:				R_TRIG;
	FD_MultiBip:				F_TRIG;
	VAR_Cpt_Bip:				USINT;
END_VAR

VAR_INPUT PERSISTENT
	PRM_Tp_Continu1:			TIME;	(*Temps bip continu 1*)
	PRM_Tp_Continu2:			TIME;	(*Temps bip continu 2*)
	PRM_Tp_Bip_Alternatif:		TIME;	(*Temps bip alternatif : 50% de ce paramètre*)
	PRM_Tp_Tempo_Alternatif:	TIME;	(*Temps d'activation du bip alternatif si PRM_Alternatif_Temporise*)
	PRM_Tp_MultiBip1:			TIME;	(*Temps un bip : 50% de ce paramètre*)
	PRM_Tp_MultiBip2:			TIME;	(*Temps pour chaque double-bip*)
	PRM_Tp_Tempo_MultiBip:		TIME;	(*Temps d'activation du double bip si PRM_DoubleBip_Temporise*)
	PRM_Alternatif_Temporise:	BOOL;	(*Activation temporisée du défaut alternatif*)
	PRM_MultiBip_Temporise:		BOOL;	(*Activation temporisée du défaut double bip*)
	PRM_Acq_Continu1:			BOOL;	(*Mode inhibé par l'acquittement*)
	PRM_Acq_Continu2:			BOOL;	(*Mode inhibé par l'acquittement*)
	PRM_Acq_Alternatif:			BOOL;	(*Mode inhibé par l'acquittement*)
	PRM_Acq_MultiBip:			BOOL;	(*Mode inhibé par l'acquittement*)
	PRM_Acq_Permanent:			BOOL;	(*Mode inhibé par l'acquittement*)
	PRM_Nb_Bip:					USINT;	(*Nb de bips mode mulitbip*)
END_VAR

(*-----------------------------------------------------BIP ALTERNATIF---------------------------------------------------*)

(*Bip pendant 50% de PRM_Tp_Alternatif si I_DEF_Alternatif actif*)
VAR_Alternatif.CONF_Period_Off		:=	PRM_Tp_Bip_Alternatif/2;
VAR_Alternatif.CONF_Period_On		:=	PRM_Tp_Bip_Alternatif/2;

(*Timer activation bip temporisé si option sélectionnée*)
TIMER_Alternatif.PT	:=	PRM_Tp_Tempo_Alternatif;
TIMER_Alternatif.IN	:=	I_DEF_Alternatif AND PRM_Alternatif_Temporise;
TIMER_Alternatif();

VAR_Alternatif(IN_On	:=	((I_DEF_Alternatif AND NOT PRM_Alternatif_Temporise) OR TIMER_Alternatif.Q) AND NOT RESET);

FM_Alternatif.CLK	:=	I_DEF_Alternatif;
FM_Alternatif();

(*-----------------------------------------------------MULTI BIP---------------------------------------------------*)

(*Multi bip de 50% de PRM_Tp_MultiBip1 toutes les PRM_Tp_MultiBip2 si I_DEF_MultiBip actif*)
VAR_MultiBip.CONF_Period_Off		:=	PRM_Tp_MultiBip1/2;
VAR_MultiBip.CONF_Period_On			:=	PRM_Tp_MultiBip1/2;

FD_MultiBip.CLK	:=	VAR_MultiBip.STATE_ON;
FD_MultiBip();
IF FD_MultiBip.Q THEN
	VAR_Cpt_Bip		:=	VAR_Cpt_Bip + 1;
END_IF
TIMER_MultiBip2.IN		:=	(VAR_Cpt_Bip = PRM_Nb_Bip);
TIMER_MultiBip2.PT		:=	PRM_Tp_MultiBip2 - REAL_TO_TIME(PRM_nb_Bip*TIME_TO_REAL(PRM_Tp_MultiBip1));
TIMER_MultiBip2();
IF TIMER_MultiBip2.Q OR NOT I_DEF_MultiBip THEN
	VAR_Cpt_Bip		:=	0;
END_IF

(*Timer activation bip temporisé si option sélectionnée*)
TIMER_MultiBip.PT	:=	PRM_Tp_Tempo_MultiBip;
TIMER_MultiBip.IN	:=	I_DEF_MultiBip AND PRM_MultiBip_Temporise;
TIMER_MultiBip();

VAR_MultiBip(IN_On	:=	((I_DEF_MultiBip AND NOT PRM_MultiBip_Temporise AND (VAR_Cpt_Bip < PRM_Nb_Bip)) OR TIMER_MultiBip.Q) AND NOT RESET);

FM_MultiBip.CLK	:=	I_DEF_MultiBip;
FM_MultiBip();

(*-----------------------------------------------------BIP CONTINU TEMPORISE 1---------------------------------------------------*)

TIMER_Continu1.PT		:=	PRM_Tp_Continu1;
TIMER_Continu1.IN		:=	I_DEF_Continu1 AND NOT RESET;
TIMER_Continu1();

FM_Continu1.CLK	:=	I_DEF_Continu1;
FM_Continu1();

(*-----------------------------------------------------BIP CONTINU TEMPORISE 2---------------------------------------------------*)

TIMER_Continu2.PT		:=	PRM_Tp_Continu2;
TIMER_Continu2.IN		:=	I_DEF_Continu2 AND NOT RESET;
TIMER_Continu2();

FM_Continu2.CLK	:=	I_DEF_Continu2;
FM_Continu2();

(*-----------------------------------------------------BIP PERMANENT---------------------------------------------------*)

FM_Permanent.CLK	:=	I_DEF_Permanent;
FM_Permanent();


(*-----------------------------------------------------SORTIE---------------------------------------------------*)
IF (FM_Permanent.Q AND PRM_Acq_Permanent)
	OR (FM_Continu1.Q AND PRM_Acq_Continu1)
	OR (FM_Continu2.Q AND PRM_Acq_Continu2)
	OR (FM_Alternatif.Q AND PRM_Acq_Alternatif)
	OR (FM_MultiBip.Q AND PRM_Acq_MultiBip) THEN
		M_ACQ				:=	FALSE;
		OUT_Buzzer			:=	TRUE;
ELSIF (I_DEF_Permanent AND (NOT PRM_Acq_Permanent OR (NOT M_ACQ AND PRM_Acq_Permanent)))
	OR (TIMER_Continu1.Q AND (NOT PRM_Acq_Continu1 OR (NOT M_ACQ AND PRM_Acq_Continu1)))
	OR (TIMER_Continu2.Q AND (NOT PRM_Acq_Continu2 OR (NOT M_ACQ AND PRM_Acq_Continu2)))
	OR (VAR_Alternatif.STATE_ON AND (NOT PRM_Acq_Alternatif OR (NOT M_ACQ AND PRM_Acq_Alternatif)))
	OR (VAR_MultiBip.STATE_ON AND (NOT PRM_Acq_MultiBip OR (NOT M_ACQ AND PRM_Acq_MultiBip)))
	THEN
		OUT_Buzzer			:=	TRUE;
ELSE
		OUT_Buzzer			:=	FALSE;
END_IF

END_FUNCTION_BLOCK

// ---- POUs/Programme/BLOCK_PRG_INFO_CLIENT.TcPOU
FUNCTION_BLOCK BLOCK_PRG_INFO_CLIENT

VAR_INPUT
END_VAR
VAR_OUTPUT
	(*sorties MOXA*)
	OUT_MOXA_O1	AT%Q*:			BOOL;
	OUT_MOXA_O2	AT%Q*:			BOOL;
	OUT_MOXA_O3	AT%Q*:			BOOL;
	OUT_MOXA_O4	AT%Q*:			BOOL;
	OUT_MOXA_O5	AT%Q*:			BOOL;
	OUT_MOXA_O6	AT%Q*:			BOOL;
	OUT_MOXA_O7	AT%Q*:			BOOL;
	OUT_MOXA_O8	AT%Q*:			BOOL;
END_VAR
VAR
END_VAR


(*COMMUNICATION CLIENT BOITIER MOXA*)

(*1 - Production : process en cours*)
OUT_MOXA_O1	:=	MACHINE.STATE_Prod;
(*2 - Réglage : Mode manuel*)
OUT_MOXA_O2	:=	MACHINE.STATE_Manu;
(*3 - Attente de chargement : Mode auto en attente de process*)
OUT_MOXA_O3	:=	MACHINE.STATE_Wait_Prod;
(*4 - Panne : Défaut présent*)
OUT_MOXA_O4	:=	MACHINE.I_def_stop OR MACHINE.I_def_inter;
(*5 - Power ON*)
OUT_MOXA_O5	:=	MACHINE.STATE_On;
(*6 - Power OFF*)
OUT_MOXA_O6	:=	MACHINE.STATE_Off;

END_FUNCTION_BLOCK

// ---- POUs/Composant/AXES/BLOCK_VARIATEUR_MOTEUR.TcPOU
FUNCTION_BLOCK BLOCK_VARIATEUR_MOTEUR

VAR_INPUT
	I_PARAM_SYSTEM_OK:			BOOL;			(*paramétrage système ok*)
(*paramètre standard*)
	RESET:   					BOOL; 			(*Condition RAZ actionneur*)
	MANUAL:  					BOOL; 			(*Mode manuel*)

	DOOR:						BOOL;			(*indicateur fermeture porte*)

(*parametre de pilotage en entrée*)
	CO_On:   					BOOL;	 		(*Ordre mode automatique activation*)
	EN_On_INT:   				BOOL:=TRUE;		(*Condition d'autorisation d'activation donnée par le bloc qui instancie le bloc actuator*)
	EN_Off_INT:  				BOOL:=TRUE;		(*Condition d'autorisation de désactivation donnée par le bloc qui instacie le bloc actuator*)
	EN_On_EXT:					BOOL:=TRUE;		(*condition d'autorisation d'activation externe*)
	EN_Off_EXT:					BOOL:=TRUE;		(*condition d'autorisation de desactivation externe*)

	IN_OK AT %I*:			BOOL;				(*Indique que le variateur est OK, pas en défaut*)

	PRM_Cons_Vitesse:		REAL;				(*consigne de vitesse du PS de 0*)

	DEF_Off_auto:			PRCDEF;		(*Défaut de désactivation automatique*)
(*	DEF_SURV_ROTATION:		PRCDEF;		(*Défaut de surveillance de la rotation*)	*)
(*	DEF_MARCHE:				PRCDEF;		(*Défaut de marche du variateur*)		*)
	DEF_Variateur:			PRCDEF;		(*Défaut indiquant que le variateur est pas ok*)

	AO_VITESSE:				ANALOG_OUTPUT;
	TIMER_OFF:				TON;
END_VAR

VAR
	M_On:  						BOOL; 										(*Ordre mode manuel activation rotation*)
	M_Off:   					BOOL; 										(*Ordre mode manuel désactivation*)
	RCP_M_On:   				BOOL;
	RCP_M_Off:  				BOOL;
	VAR_On:						BOOL;										(*variable intermédiaire avant affectation de la sortie OUT_On *)
	VAR_Off:					BOOL;										(*Variable intermédiaire avant affectation de la sortie OUT_Off *)
	TIMER_DOOR_CLOSED:	TON;
	VAR_TIM_SURV:			TIME;
	AI_POT: BOOL;
END_VAR

VAR_INPUT PERSISTENT
(*Entité*)
	IsComponent:			BOOL;		(*entité : composant*)
	IdXML:					STRING;		(*nom entité : identifiant pour recherche dans dico*)
	TagXML:					UINT;		(*nom entité : identifiant pour recherche dans dico*)
	IdParent:				STRING;		(*MNEMO de l'appelant*)
	MNEMO:					STRING;		(*MNEMO de l'entité*)
	CONF_MAX_RPM:			REAL;		(*Vitesse maximum en unité physique*)
	CONF_EN_On:				USINT:=0;	(*définit la réaction du système en cas de perte des conditions d'autorisation d'activation EN_On*)
										(* 0 = désactivation automatique  en cas de perte des conditions d'autorisation d'activation uniquement en manuel*)
										(* 1 = désactivation automatique en cas de perte des conditions d'autorisation d'activation en auto et en manuel*)
										(* 2 = Pas de déscativation automatique*)
	CONF_No_Safety_Auto:	BOOL:=FALSE;
										(*option de desactivation des conditions d'autorisation en mode automatique*)
	TIMER_RETARD_SURV : TON;
END_VAR

VAR_OUTPUT

	OUT_MPS11 				AT %Q*:	BOOL;							(*SORTIE TOR ROTATION PS *)
	STATE_Consigne:			REAL;									(*Consigne de vitesse de rotation appliquée*)
	STATE_On:	   			BOOL; 									(*Indicateur moteur en marche*)
	STATE_Off:				BOOL;									(*Indicateur moteur à l'arrêt*)
	STATE_Nok:				BOOL;									(*Etat non ok*)
	AUTOR_On_IHM:			BOOL; 									(*etat activation autorisée depuis la supervision*)
	AUTOR_Off_IHM:			BOOL; 									(*etat désactivation autorisée depuis la supervision*)
	AUTOR_On_PLC:			BOOL;									(*etat activation autorisée depuis l'automate*)
	AUTOR_Off_PLC:			BOOL;									(*etat désactivation autorisée depuis l'automate*)
	OUT_QVMPS11 			AT %Q*: INT;								(*consigne de vitesse appliquée au moteur*)
END_VAR

	IdXML:= '5';
	TagXML:= 2;
	DEF_OFF_AUTO.IdXML := '3';
	DEF_OFF_AUTO.TagXML :=10;
	(*DEF_MARCHE.IdXML := '3';
	DEF_MARCHE.TagXML:=1;*)
	DEF_Variateur.IdXML	:= '5';
	DEF_Variateur.TagXML	:= 15;

(* Réception des ordres en mode manuel*)
	RCP_M_On	 		:=	M_On;
	RCP_M_Off			:=	M_Off;

(*Autorisation*)
	AUTOR_On_IHM		:= 	MANUAL AND ((EN_On_INT AND EN_On_EXT AND DOOR)
							OR MANUAL_SAFETY_OFF) AND NOT RESET AND NOT VAR_On;
	AUTOR_Off_IHM		:= 	MANUAL AND ((EN_Off_INT AND EN_Off_EXT)  OR
							MANUAL_SAFETY_OFF) AND NOT RESET;
	AUTOR_On_PLC		:=	 NOT MANUAL AND ((EN_On_INT AND EN_On_EXT AND DOOR)
							OR CONF_No_Safety_Auto) AND NOT RESET;
	AUTOR_Off_PLC		:= 	NOT MANUAL AND ((EN_Off_INT AND EN_Off_EXT)
							OR CONF_No_Safety_Auto) AND NOT RESET;

(*defaut desactivation automatique*)
	DEF_Off_Auto.CONDITION :=        (NOT EN_On_INT OR NOT EN_On_EXT OR NOT DOOR)
								AND  VAR_On
								AND ((CONF_En_ON=1) OR ((CONF_EN_On=0) AND MANUAL))
								AND NOT RESET;
	DEF_Off_auto.DELAY:=T#0ms;
	DEF_Off_Auto();

(*gestion des sorties*)
IF 		(RCP_M_On AND AUTOR_On_IHM) OR
		(CO_On AND AUTOR_On_PLC)	THEN
				VAR_On		:= 	TRUE;
				VAR_Off			:= 	FALSE;
ELSIF
		(RCP_M_Off AND AUTOR_Off_IHM)  OR
	    	(NOT CO_On AND AUTOR_Off_PLC)
		OR RESET OR DEF_Off_Auto.DEF THEN
				VAR_On		:=	FALSE;
				VAR_Off			:=	TRUE;		(*COR_MOMO*)
END_IF;

OUT_MPS11		:=	VAR_On ;		(*Affectation de la sortie rotation PS*)

STATE_On:= 	OUT_MPS11 ;
TIMER_OFF.IN :=  NOT OUT_MPS11;
TIMER_OFF(PT:=T#45s);	(*Temporisation de validation de l'arrêt du PS*)
STATE_OFF:=	TIMER_OFF.Q;

(*Conversion de la valeur analogique*)
AO_VITESSE.Value := PRM_Cons_Vitesse;		(*Consigne 0-10v*)

AO_VITESSE(
	CONF_Max:= CONF_MAX_RPM,
	CONF_Min:= 0.0,
	CONF_Bipolar:=FALSE,
	CONF_Range:=1.0,
	Value:=  ,
	OUTPUT=> OUT_QVMPS11);

(*
DEF_MARCHE.CONDITION 		:=	STATE_On AND NOT IN_OK;
DEF_MARCHE.DELAY				:=	T#5s;
DEF_MARCHE;
*)
DEF_Variateur.CONDITION		:=	NOT IN_OK AND NOT RESET;
DEF_Variateur.DELAY		:= T#5s;
DEF_Variateur();

STATE_NOK:=	DEF_Off_AUTO.DEF OR DEF_Variateur.DEF;

(* Reset des ordres *)
IF M_On AND RCP_M_On THEN
	M_On 	:= FALSE;
END_IF;
IF M_Off AND RCP_M_Off THEN
	M_Off		 := FALSE;
END_IF;

END_FUNCTION_BLOCK

// ---- POUs/Composant/EVAP/BLOCK_IND_CREUSET_GENIUS.TcPOU
(*Gestion d'un indexeur de creuset par le contrôleur GENIUS*)
(*Changement de position dés modification de la consigne*)
(*Mode Ferrotec*)

(****************historique des versions*****************************)

(* Version 1-0 - Sezai - VERSION INIITIALE - 8152*)
(* Version 2-0 - GV - Modification gestion des sorties pour gestion 8 creusets - 10315 - EVA451 n°20*)

(*************************************************************************)

FUNCTION_BLOCK BLOCK_IND_CREUSET_GENIUS

VAR_INPUT
	RESET:			 				BOOL;
	PRM_NCR:						USINT:=1;		(*Commande de position*)
	PRM_NBAL:						USINT:=1;		(*Numéro de balayage*)
	IN_POS_OK  		AT %I* :		BOOL;			(*Etat indexeur sur creuset selectionné*)
	I_FIL_ON:						BOOL;			(*interlock source en marche*)
	DEF_POSITIONNEMENT:				PRCDEF;			(*Défaut de positionnement*)
	IN_POWER:						REAL;			(*Puissance appliquée au creuset*)
END_VAR

VAR
	VAR_WORD_CR:				WORD;
	VAR_WORD_SW:				WORD;

	FM_POS_OK:					R_TRIG;									(*Front montant de position ok*)

	VAR_Cpt_Temps_C1: 			BLOCK_CPT_TEMPS;						(*Compteur de fonctionnement creuset 1*)
	VAR_Cpt_Temps_C2: 			BLOCK_CPT_TEMPS;						(*Compteur de fonctionnement creuset 2*)
	VAR_Cpt_Temps_C3: 			BLOCK_CPT_TEMPS;						(*Compteur de fonctionnement creuset 3*)
	VAR_Cpt_Temps_C4: 			BLOCK_CPT_TEMPS;						(*Compteur de fonctionnement creuset 4*)
	VAR_Cpt_Temps_C5: 			BLOCK_CPT_TEMPS;						(*Compteur de fonctionnement creuset 5*)
	VAR_Cpt_Temps_C6: 			BLOCK_CPT_TEMPS;						(*Compteur de fonctionnement creuset 6*)
	VAR_Cpt_Temps_C7: 			BLOCK_CPT_TEMPS;						(*Compteur de fonctionnement creuset 7*)
	VAR_Cpt_Temps_C8: 			BLOCK_CPT_TEMPS;						(*Compteur de fonctionnement creuset 8*)

END_VAR
VAR_OUTPUT

	OUT_POS_CR1 AT %Q*:			BOOL;		(*position de l'indexeur  OUT_POS_CRx*)
	OUT_POS_CR2 AT %Q*:			BOOL;
	OUT_POS_CR3 AT %Q*:			BOOL;
	OUT_POS_CR4 AT %Q*:			BOOL;
	OUT_POS_CR5 AT %Q*:			BOOL;
	OUT_POS_CR6 AT %Q*:			BOOL;
	STATE_POS_CR:				USINT;
	STATE_ROT:					BOOL;		(*Creuset en rotation*)
	STATE_NOK:					BOOL;
	STATE_POS_OK:				BOOL;
	STATE_MAT:					STRING;
END_VAR

VAR_INPUT PERSISTENT
	CONF_NCR:					INT:=6;					(*nombre de creuset de la source*)
	PRM_MAT: 					ARRAY[0..8] OF STRING;	(*nom de la matière associée au creuset*)
	VAR_MEM_CR:					USINT;					(*Mémoire numéro de creuset utilisé*)
	VAR_MEM_SW:					USINT;					(*Mémoire numéri de balayage utilisé*)

	(*Entité*)
	IsComponent:		BOOL;			(*entité : composant*)
	IdXML:				STRING;			(*nom entité : identifiant pour recherche dans dico*)
	TagXML:				UINT;			(*nom entité : identifiant pour recherche dans dico*)
	IdParent:			STRING;			(*MNEMO de l'appelant*)
	MNEMO:				STRING;			(*MNEMO de l'entité*)
END_VAR

(*Défaut*)
DEF_POSITIONNEMENT.IdXml		:=	'14';
DEF_POSITIONNEMENT.TagXml		:=	2;

(*memorisation de la consigne du creuset*)
IF ( NOT ( CONF_NCR = 1))
	AND (VAR_MEM_CR <> PRM_NCR)	 THEN
	VAR_MEM_CR := PRM_NCR;
	(* RAZ defaut positionnement*)
	DEF_POSITIONNEMENT.CONDITION := FALSE;
	DEF_POSITIONNEMENT();
	STATE_POS_CR := 0;	(* pas de position determinée*)
END_IF

(*memorisation de la consigne de balayage*)
IF (VAR_MEM_SW <> PRM_NBAL) THEN
	VAR_MEM_SW := PRM_NBAL;
END_IF


FM_POS_OK(CLK:= IN_POS_OK);
(* sur front montant si multi creuset*)
IF FM_POS_OK.Q AND (CONF_NCR > 1) THEN
	STATE_POS_CR := VAR_MEM_CR;
END_IF

VAR_WORD_CR := VAR_MEM_CR - 1;
VAR_WORD_SW := VAR_MEM_SW - 1;

(*Parametrage des positions*)
OUT_POS_CR1:=	VAR_WORD_CR.0;
OUT_POS_CR2:=	VAR_WORD_CR.1;
OUT_POS_CR3:=	VAR_WORD_CR.2;
OUT_POS_CR4:=	VAR_WORD_SW.0;
OUT_POS_CR5:=	VAR_WORD_SW.1;
OUT_POS_CR6:=	VAR_WORD_SW.2;

DEF_POSITIONNEMENT.CONDITION := NOT ( STATE_POS_CR = VAR_MEM_CR) AND NOT (CONF_NCR = 1);
DEF_POSITIONNEMENT.DELAY := T#120s;
DEF_POSITIONNEMENT();


(*gestion compteur d'utilisation*)
(*creuset 1*)
VAR_Cpt_Temps_C1.I_On := (STATE_POS_CR = 1) AND I_FIL_ON;
VAR_Cpt_Temps_C1.TagXML := 11;
VAR_Cpt_Temps_C1();

(*creuset 2*)
VAR_Cpt_Temps_C2.I_On := (STATE_POS_CR = 2) AND I_FIL_ON;
VAR_Cpt_Temps_C2.TagXML := 12;
VAR_Cpt_Temps_C2();

(*creuset 3*)
VAR_Cpt_Temps_C3.I_On := (STATE_POS_CR = 3) AND I_FIL_ON;
VAR_Cpt_Temps_C3.TagXML := 13;
VAR_Cpt_Temps_C3();

(*creuset 4*)
VAR_Cpt_Temps_C4.I_On := (STATE_POS_CR = 4) AND I_FIL_ON;
VAR_Cpt_Temps_C4.TagXML := 14;
VAR_Cpt_Temps_C4();

(*creuset 5*)
VAR_Cpt_Temps_C5.I_On := (STATE_POS_CR = 5) AND I_FIL_ON;
VAR_Cpt_Temps_C5.TagXML := 15;
VAR_Cpt_Temps_C5();

(*creuset 6*)
VAR_Cpt_Temps_C6.I_On := (STATE_POS_CR = 6) AND I_FIL_ON;
VAR_Cpt_Temps_C6.TagXML := 16;
VAR_Cpt_Temps_C6();

(*creuset 7*)
VAR_Cpt_Temps_C7.I_On := (STATE_POS_CR = 7) AND I_FIL_ON;
VAR_Cpt_Temps_C7.TagXML := 17;
VAR_Cpt_Temps_C7();

(*creuset 8*)
VAR_Cpt_Temps_C8.I_On := (STATE_POS_CR = 8) AND I_FIL_ON;
VAR_Cpt_Temps_C8.TagXML := 18;
VAR_Cpt_Temps_C8();
(**)

STATE_NOK:= DEF_POSITIONNEMENT.DEF;
STATE_POS_OK := NOT (STATE_POS_CR = 0);

IF STATE_POS_CR > 0 AND STATE_POS_CR <=8 THEN
	STATE_MAT:= PRM_MAT[STATE_POS_CR];
ELSE
	STATE_MAT:= '';
END_IF

END_FUNCTION_BLOCK

// ---- POUs/Composant/EVAP/BLOCK_IND_CR_379_TELEMARK_V4.TcPOU
FUNCTION_BLOCK BLOCK_IND_CR_379_TELEMARK_V4

(* Pour utilisation d'un indexeur de creuset telemark 379 à 6 creusets max *)

(****************historique des versions*****************************)

(* Version 0 - 05/01/12 - JPC *)
(* Version 1 - 01/15 - GV - Adaptation pour journal des évenements + Ajout compteurs d'utilisation + Ajout Co_Change + M_Change *)
(* Version 2 - 07/15 - GV - Ajout temporisation pour obtention STATE_POS_OK*)
(* Version 3 - 09/22 - GV - Ajout condition d'inhibition des défauts*)
(* Version 4 - 11/23 - HG - Inhibition défaut positionnement si aucune sortie activée
							Modif State_pos en fonction de tous les retours
							Ajout gestion remote, indispensable sur sortie mode éco-veille*)
(*************************************************************************)

VAR_INPUT
	MANUAL:					BOOL;		(*Mode de pilotage manuel *)
	RESET:					BOOL;		(*Condition de réiinitialisation de la fonction *)

	CO_Change:				BOOL;		(*Demande de changement de creuset en automatique*)
	CO_Remote:				BOOL;		(*Demande d'activation du mode remote en automatique*)

	I_FIL_ON:				BOOL;
	PRM_NCR:				USINT:=1;	(*Commande de position*)

	IN_POWER:				REAL;		(*Puissance appliquée au creuset*)

	IN_POS1:				BOOL;		(*position de l'indexeur*)
	IN_POS2:				BOOL;
	IN_POS3:				BOOL;
	IN_POS4:				BOOL;		(*position de l'indexeur*)
	IN_POS5:				BOOL;
	IN_POS6:				BOOL;

	DEF_POSITIONNEMENT:	PRCDEF;	(*Défaut de positionnement*)
	I_Inhibe_Def:		BOOL;	(*Inhibition des défauts*)
END_VAR

VAR
	VAR_Cpt_Temps:				ARRAY[0..6] OF BLOCK_CPT_TEMPS;		(*Compteur de fonctionnement pour chaque creuset*)
	VAR_Cpt_Puissance:			ARRAY[0..6] OF BLOCK_CPT_INTEG;		(*Compteur pour chaque creuset*)
	VAR_Cpt_Epaisseur:			ARRAY[0..6] OF BLOCK_CPT_INTEG;		(*Compteur d'épaisseur pour chaque creuset*)
	I:							USINT;									(*Variable d'itération*)

	M_Change:					BOOL;	(* Ordre de changement de creuset en manuel *)
	RCP_M_Change:				BOOL;	(* Bit de reception de l'ordre de Marche/Arrêt du module de balayage *)
	VAR_Change:					BOOL;	(* Variable intermédiaire de marche du module de balayage*)
	M_Remote:					BOOL;	(* Ordre de changement commande remote *)
	RCP_M_Remote:				BOOL;	(* Bit de reception de l'ordre de remote du module de balayage*)
	VAR_Remote:					BOOL;	(* Variable intermédiaire commande remote du module de balayage*)

	TIMER_Valid_Pos_Creuset:		TON;	(*Attentede validation du positionnement du creuset*)
END_VAR

VAR_OUTPUT
	AUTOR_Change_IHM:			BOOL;		(*indique que le changement de creuset est autorisé en mode manuel depuis l'IHM*)
	AUTOR_Change_PLC:			BOOL;		(*indique que le changement de creuset est autorisé en mode automatique depuis l'automate*)
	AUTOR_Remote_IHM:			BOOL;		(*indique que le changement mode remote est autorisé en mode manuel depuis l'IHM*)
	AUTOR_Remote_PLC:			BOOL;		(*indique que le changement more remote est autorisé en mode automatique depuis l'automate*)
	
	OUT_SEL1:					BOOL;		(*sélection  des creusets*)
	OUT_SEL2:					BOOL;
	OUT_SEL3:					BOOL;
	OUT_SEL4:					BOOL;		(*sélection  des creusets *)
	OUT_SEL5:					BOOL;
	OUT_SEL6:					BOOL;
	OUT_RMT:					BOOL;		(*pilotage remote*)
	STATE_ROT:					BOOL;		(*Creuset en rotation*)
	STATE_NOK:					BOOL;		(*Positionnement nok*)
	STATE_POS_OK:				BOOL;		(*Positionnement ok*)
	STATE_POS:					USINT;
	STATE_MAT:					STRING;
END_VAR

VAR_INPUT PERSISTENT
	CONF_NCR:		USINT;	(*Nombre de creuset disponible*)

	PRM_MAT: 		ARRAY[0..8] OF STRING;		(*nom de la matière associée au creuset*)

	(*Entité*)
	IsComponent:		BOOL;			(*entité : composant*)
	IdXML:				STRING;			(*nom entité : identifiant pour recherche dans dico*)
	TagXML:				UINT;			(*nom entité : identifiant pour recherche dans dico*)
	IdParent:			STRING;			(*MNEMO de l'appelant*)
	MNEMO:				STRING;			(*MNEMO de l'entité*)
END_VAR

(*Défaut*)
DEF_POSITIONNEMENT.IdXml		:=	'14';
DEF_POSITIONNEMENT.TagXml		:=	2;

(* Gestion des ordres en mode manuel *)
RCP_M_Change			:=	M_Change;
RCP_M_Remote			:=	M_Remote;

(*gestion des bits d'autorisation en mode manuel*)
AUTOR_Change_IHM		:=	NOT RESET AND NOT Var_Change AND NOT I_FIL_ON AND MANUAL;
AUTOR_Change_PLC		:=	NOT RESET AND NOT I_FIL_ON AND NOT MANUAL;
AUTOR_Remote_IHM		:=	NOT RESET AND MANUAL;
AUTOR_Remote_PLC		:=	NOT RESET AND NOT MANUAL;

(*gestion des variables intermédiare*)
(*Changement Creuset*)
IF	(CO_Change AND AUTOR_Change_PLC)
		 OR 	( RCP_M_Change AND AUTOR_Change_IHM) THEN
			VAR_Change 		:= 	TRUE;
ELSIF (VAR_Change AND STATE_POS_OK) THEN
			VAR_Change		:=	FALSE;
END_IF;
(*Remote*)
IF	(CO_Remote AND AUTOR_Remote_PLC)
		 OR 	(RCP_M_Remote AND NOT VAR_Remote AND AUTOR_Remote_IHM) THEN
			VAR_Remote 		:= 	TRUE;
ELSIF (NOT CO_Remote AND NOT RESET AND NOT MANUAL)
		OR 	(RCP_M_Remote AND VAR_Remote AND AUTOR_Remote_IHM)
		OR 	RESET THEN
			VAR_Remote		:=	FALSE;
END_IF;

IF PRM_NCR > CONF_NCR THEN
	PRM_NCR := CONF_NCR;
END_IF

IF VAR_Change THEN
	CASE PRM_NCR OF
			6:
				OUT_SEL1 := FALSE;
				OUT_SEL2 := FALSE;
				OUT_SEL3 := FALSE;
				OUT_SEL4 := FALSE;
				OUT_SEL5 := FALSE;
				OUT_SEL6 := TRUE;
			5:
				OUT_SEL1 := FALSE;
				OUT_SEL2 := FALSE;
				OUT_SEL3 := FALSE;
				OUT_SEL4 := FALSE;
				OUT_SEL5 := TRUE;
				OUT_SEL6 := FALSE;
			4:
				OUT_SEL1 := FALSE;
				OUT_SEL2 := FALSE;
				OUT_SEL3 := FALSE;
				OUT_SEL4 := TRUE;
				OUT_SEL5 := FALSE;
				OUT_SEL6 := FALSE;
			3:
				OUT_SEL1 := FALSE;
				OUT_SEL2 := FALSE;
				OUT_SEL3 := TRUE;
				OUT_SEL4 := FALSE;
				OUT_SEL5 := FALSE;
				OUT_SEL6 := FALSE;
			2:
				OUT_SEL1 := FALSE;
				OUT_SEL2 := TRUE;
				OUT_SEL3 := FALSE;
				OUT_SEL4 := FALSE;
				OUT_SEL5 := FALSE;
				OUT_SEL6 := FALSE;
			1:
				OUT_SEL1 := TRUE;
				OUT_SEL2 := FALSE;
				OUT_SEL3 := FALSE;
				OUT_SEL4 := FALSE;
				OUT_SEL5 := FALSE;
				OUT_SEL6 := FALSE;
	END_CASE;
END_IF
OUT_RMT	:=	VAR_Remote;

IF IN_POS1 AND NOT IN_POS2 AND NOT IN_POS3 AND NOT IN_POS4 AND NOT IN_POS5 AND NOT IN_POS6 THEN
		STATE_POS := 1;
ELSIF IN_POS2 AND NOT IN_POS1 AND NOT IN_POS3 AND NOT IN_POS4 AND NOT IN_POS5 AND NOT IN_POS6 THEN
		STATE_POS := 2;
ELSIF IN_POS3 AND NOT IN_POS1 AND NOT IN_POS2 AND NOT IN_POS4 AND NOT IN_POS5 AND NOT IN_POS6 THEN
		STATE_POS := 3 ;
ELSIF IN_POS4 AND NOT IN_POS1 AND NOT IN_POS2 AND NOT IN_POS3 AND NOT IN_POS5 AND NOT IN_POS6 THEN
		STATE_POS := 4;
ELSIF IN_POS5 AND NOT IN_POS1 AND NOT IN_POS2 AND NOT IN_POS3 AND NOT IN_POS4 AND NOT IN_POS6 THEN
		STATE_POS := 5;
ELSIF IN_POS6 AND NOT IN_POS1 AND NOT IN_POS2 AND NOT IN_POS3 AND NOT IN_POS4 AND NOT IN_POS5 THEN
		STATE_POS := 6;
END_IF;

(*Attente de validation positionnement creuset*)
TIMER_Valid_Pos_Creuset.IN	:=	(IN_POS1 = OUT_SEL1) AND (IN_POS2 = OUT_SEL2) AND (IN_POS3 = OUT_SEL3) AND
								(IN_POS4 = OUT_SEL4) AND (IN_POS5 = OUT_SEL5) AND (IN_POS6 = OUT_SEL6);
TIMER_Valid_Pos_Creuset(PT:=T#500ms);
STATE_POS_OK	:= TIMER_Valid_Pos_Creuset.Q;


STATE_ROT:=	((IN_POS1 <> OUT_SEL1) OR ( IN_POS2 <> OUT_SEL2) OR (IN_POS3 <> OUT_SEL3 ) OR
				(IN_POS4 <> OUT_SEL4) OR (IN_POS5 <> OUT_SEL5) OR (IN_POS6 <> OUT_SEL6));

DEF_POSITIONNEMENT.CONDITION :=  ((IN_POS1 <> OUT_SEL1) OR ( IN_POS2 <> OUT_SEL2) OR (IN_POS3 <> OUT_SEL3 ) OR
										 (IN_POS4 <> OUT_SEL4) OR (IN_POS5 <> OUT_SEL5) OR (IN_POS6 <> OUT_SEL6)) 
									AND NOT I_Inhibe_Def AND NOT (NOT OUT_SEL1 AND NOT OUT_SEL2 AND NOT OUT_SEL3 AND NOT OUT_SEL4);
DEF_POSITIONNEMENT.DELAY := T#180S;
DEF_POSITIONNEMENT();

(*gestion compteur d'utilisation*)
FOR I := 1 TO 6 BY 1 DO
	VAR_Cpt_Puissance[I].CONF_Coeff:=1;
	VAR_Cpt_Puissance[I].CONF_TimeUnit:=2;
	VAR_Cpt_Puissance[I].I_Value := IN_POWER;
	VAR_Cpt_Puissance[I].I_On := (STATE_POS = I);
	VAR_Cpt_Puissance[I]();

	VAR_Cpt_Temps[I].I_On := (STATE_POS = I) AND I_FIL_ON;		(*Compteur d'utilisation des creusets*)
	VAR_Cpt_Temps[I]();
END_FOR

STATE_NOK:= DEF_POSITIONNEMENT.DEF;

IF STATE_POS > 0 AND STATE_POS <= CONF_NCR THEN
	STATE_MAT:= PRM_MAT[STATE_POS];
ELSE
	STATE_MAT:= '';
END_IF

(* Reset des ordres*)
IF M_Change	AND RCP_M_Change THEN
	M_Change			:=	FALSE;
END_IF
IF M_Remote	AND RCP_M_Remote THEN
	M_Remote			:=	FALSE;
END_IF

END_FUNCTION_BLOCK

// ---- POUs/Composant/EVAP/BLOCK_IND_CR_379_TELEMARK_V3.TcPOU
FUNCTION_BLOCK BLOCK_IND_CR_379_TELEMARK_V3

(* Pour utilisation d'un indexeur de creuset telemark 379 à 6 creusets max *)

(****************historique des versions*****************************)

(* Version 0 - 05/01/12 - JPC *)
(* Version 1 - 01/15 - GV - Adaptation pour journal des évenements + Ajout compteurs d'utilisation + Ajout Co_Change + M_Change *)
(* Version 2 - 07/15 - GV - Ajout temporisation pour obtention STATE_POS_OK*)
(* Version 3 - 09/22 - GV - Ajout condition d'inhibition des défauts*)

(*************************************************************************)

VAR_INPUT
	MANUAL:					BOOL;		(*Mode de pilotage manuel *)
	RESET:					BOOL;		(*Condition de réiinitialisation de la fonction *)

	CO_Change:				BOOL;		(*Demande de changement de creuset en automatique*)

	I_FIL_ON:				BOOL;
	PRM_NCR:				USINT:=1;	(*Commande de position*)

	IN_POWER:				REAL;		(*Puissance appliquée au creuset*)

	IN_POS1:				BOOL;		(*position de l'indexeur*)
	IN_POS2:				BOOL;
	IN_POS3:				BOOL;
	IN_POS4:				BOOL;		(*position de l'indexeur*)
	IN_POS5:				BOOL;
	IN_POS6:				BOOL;

	DEF_POSITIONNEMENT:	PRCDEF;	(*Défaut de positionnement*)
	I_Inhibe_Def:		BOOL;	(*Inhibition des défauts*)
END_VAR

VAR
	VAR_Cpt_Temps:				ARRAY[0..6] OF BLOCK_CPT_TEMPS;		(*Compteur de fonctionnement pour chaque creuset*)
	VAR_Cpt_Puissance:			ARRAY[0..6] OF BLOCK_CPT_INTEG;		(*Compteur pour chaque creuset*)
	VAR_Cpt_Epaisseur:			ARRAY[0..6] OF BLOCK_CPT_INTEG;		(*Compteur d'épaisseur pour chaque creuset*)
	I:							USINT;									(*Variable d'itération*)

	M_Change:					BOOL;	(* Ordre de changement de creuset en manuel *)
	RCP_M_Change:				BOOL;	(* Bit de reception de l'ordre de Marche/Arrêt du module de balayage *)
	VAR_Change:					BOOL;	(* Variable intermédiaire de marche du module de balayage*)

	TIMER_Valid_Pos_Creuset:		TON;	(*Attentede validation du positionnement du creuset*)
END_VAR

VAR_OUTPUT
	AUTOR_Change_IHM:			BOOL;		(*indique que le changement de creuset est autorisée en mode manuel depuis l'IHM*)
	AUTOR_Change_PLC:			BOOL;		(*indique que le changement de creuset est autorisée en mode automatique depuis l'automate*)

	OUT_SEL1:					BOOL;		(*sélection  des creusets*)
	OUT_SEL2:					BOOL;
	OUT_SEL3:					BOOL;
	OUT_SEL4:					BOOL;		(*sélection  des creusets *)
	OUT_SEL5:					BOOL;
	OUT_SEL6:					BOOL;
	STATE_ROT:					BOOL;		(*Creuset en rotation*)
	STATE_NOK:					BOOL;		(*Positionnement nok*)
	STATE_POS_OK:				BOOL;		(*Positionnement ok*)
	STATE_POS:					USINT;
	STATE_MAT:					STRING;
END_VAR

VAR_INPUT PERSISTENT
	CONF_NCR:		USINT;	(*Nombre de creuset disponible*)

	PRM_MAT: 		ARRAY[0..8] OF STRING;		(*nom de la matière associée au creuset*)

	(*Entité*)
	IsComponent:		BOOL;			(*entité : composant*)
	IdXML:				STRING;			(*nom entité : identifiant pour recherche dans dico*)
	TagXML:				UINT;			(*nom entité : identifiant pour recherche dans dico*)
	IdParent:			STRING;			(*MNEMO de l'appelant*)
	MNEMO:				STRING;			(*MNEMO de l'entité*)
END_VAR

(*Défaut*)
DEF_POSITIONNEMENT.IdXml		:=	'14';
DEF_POSITIONNEMENT.TagXml		:=	2;

(* Gestion des ordres en mode manuel *)
	RCP_M_Change			:=	M_Change;

(*gestion des bits d'autorisation en mode manuel*)
	AUTOR_Change_IHM		:=	NOT RESET AND NOT Var_Change AND NOT I_FIL_ON AND MANUAL;
	AUTOR_Change_PLC		:=	NOT RESET AND NOT I_FIL_ON AND NOT MANUAL;

(*gestion des variables intermédiare*)
(*Changement Creuset*)
	IF	(CO_Change AND AUTOR_Change_PLC)
			 OR 	( RCP_M_Change AND AUTOR_Change_IHM) THEN
				Var_Change 		:= 	TRUE;
	ELSIF (VAR_Change AND STATE_POS_OK) THEN
				Var_Change		:=	FALSE;
	END_IF;

IF PRM_NCR > CONF_NCR THEN
	PRM_NCR := CONF_NCR;
END_IF

IF VAR_Change THEN
	CASE PRM_NCR OF
			6:
				OUT_SEL1 := FALSE;
				OUT_SEL2 := FALSE;
				OUT_SEL3 := FALSE;
				OUT_SEL4 := FALSE;
				OUT_SEL5 := FALSE;
				OUT_SEL6 := TRUE;
			5:
				OUT_SEL1 := FALSE;
				OUT_SEL2 := FALSE;
				OUT_SEL3 := FALSE;
				OUT_SEL4 := FALSE;
				OUT_SEL5 := TRUE;
				OUT_SEL6 := FALSE;
			4:
				OUT_SEL1 := FALSE;
				OUT_SEL2 := FALSE;
				OUT_SEL3 := FALSE;
				OUT_SEL4 := TRUE;
				OUT_SEL5 := FALSE;
				OUT_SEL6 := FALSE;
			3:
				OUT_SEL1 := FALSE;
				OUT_SEL2 := FALSE;
				OUT_SEL3 := TRUE;
				OUT_SEL4 := FALSE;
				OUT_SEL5 := FALSE;
				OUT_SEL6 := FALSE;
			2:
				OUT_SEL1 := FALSE;
				OUT_SEL2 := TRUE;
				OUT_SEL3 := FALSE;
				OUT_SEL4 := FALSE;
				OUT_SEL5 := FALSE;
				OUT_SEL6 := FALSE;
			1:
				OUT_SEL1 := TRUE;
				OUT_SEL2 := FALSE;
				OUT_SEL3 := FALSE;
				OUT_SEL4 := FALSE;
				OUT_SEL5 := FALSE;
				OUT_SEL6 := FALSE;
	END_CASE;
END_IF

IF IN_POS1 THEN
		STATE_POS := 1;
ELSIF IN_POS2 THEN
		STATE_POS := 2;
ELSIF IN_POS3 THEN
		STATE_POS := 3 ;
ELSIF IN_POS4 THEN
		STATE_POS := 4;
ELSIF IN_POS5 THEN
		STATE_POS := 5;
ELSIF IN_POS6 THEN
		STATE_POS := 6;
END_IF;

(*Attente de validation positionnement creuset*)
TIMER_Valid_Pos_Creuset.IN	:=	(IN_POS1 = OUT_SEL1) AND (IN_POS2 = OUT_SEL2) AND (IN_POS3 = OUT_SEL3) AND
								(IN_POS4 = OUT_SEL4) AND (IN_POS5 = OUT_SEL5) AND (IN_POS6 = OUT_SEL6);
TIMER_Valid_Pos_Creuset(PT:=T#500ms);
STATE_POS_OK	:= TIMER_Valid_Pos_Creuset.Q;


STATE_ROT:=	(IN_POS1 <> OUT_SEL1) OR ( IN_POS2 <> OUT_SEL2) OR (IN_POS3 <> OUT_SEL3 ) OR
				(IN_POS4 <> OUT_SEL4) OR (IN_POS5 <> OUT_SEL5) OR (IN_POS6 <> OUT_SEL6);

DEF_POSITIONNEMENT.CONDITION :=  ((IN_POS1 <> OUT_SEL1) OR ( IN_POS2 <> OUT_SEL2) OR (IN_POS3 <> OUT_SEL3 ) OR
										 (IN_POS4 <> OUT_SEL4) OR (IN_POS5 <> OUT_SEL5) OR (IN_POS6 <> OUT_SEL6)) AND NOT I_Inhibe_Def;
DEF_POSITIONNEMENT.DELAY := T#180s;
DEF_POSITIONNEMENT();

(*gestion compteur d'utilisation*)
FOR I := 1 TO 6 BY 1 DO
	VAR_Cpt_Puissance[I].CONF_Coeff:=1;
	VAR_Cpt_Puissance[I].CONF_TimeUnit:=2;
	VAR_Cpt_Puissance[I].I_Value := IN_POWER;
	VAR_Cpt_Puissance[I].I_On := (STATE_POS = I);
	VAR_Cpt_Puissance[I]();

	VAR_Cpt_Temps[I].I_On := (STATE_POS = I) AND I_FIL_ON;		(*Compteur d'utilisation des creusets*)
	VAR_Cpt_Temps[I]();
END_FOR

STATE_NOK:= DEF_POSITIONNEMENT.DEF;

IF STATE_POS > 0 AND STATE_POS <= CONF_NCR THEN
	STATE_MAT:= PRM_MAT[STATE_POS];
ELSE
	STATE_MAT:= '';
END_IF

(* Reset des ordres*)
IF M_Change	AND RCP_M_Change THEN
	M_Change			:=	FALSE;
END_IF

END_FUNCTION_BLOCK

// ---- POUs/Composant/EVAP/BLOCK_SOURCE_GENIUS.TcPOU
FUNCTION_BLOCK BLOCK_SOURCE_GENIUS

(****************historique des versions*****************************)

(* Version 1-0 - Sezai - VERSION INIITIALE - 8152*)
(* Version 2-0 - GV - 10/2017 - Modification HV en BLOCK_ACTUATOR pour gerer les défauts d'arrêt/marche + Modification pour être sur que l'on a un retour de courant avant de considérer en marche *)
(* Version 2-1 - GV - 09/2018 - Ajout gestion perte brève du retour IN_HV_ON*)

(*************************************************************************)

VAR_INPUT
	DOOR:					BOOL;		(*porte fermée*)
	VAC:					BOOL;		(*sécurité vide*)
	WATER:					BOOL;		(*refroidissement source ok*)
	MANUAL:					BOOL;		(*demande mode manuel*)
	I_CR_OK:				BOOL;		(*Positionnement creuset ok*)
	RESET:					BOOL;		(*reset*)

	HV:						BLOCK_ACTUATOR;		(*Source HT*)

	IN_HVON		AT%I*:		BOOL;	(*Etat Source HT en marche*)
	IN_ERROR	AT%I*:		BOOL;	(*Etat d'erreur du Genius*)

	IN_HVQ		AT%I*:		INT;		(*Entrée analogique Haute Tension source*)
	IN_FILQ		AT%I*:		INT;		(*Entrée analogique Courant filament*)


	AI_HV:			ANALOG_INPUT;
	AI_FIL:			ANALOG_INPUT;

	I_POWER:			REAL;		(*consigne de puissance appliquée en mode automatique*)
	PRM_POWER:			REAL;		(*Consigne de puissance appliquée en mode manuel*)
	CO_SRC:				BOOL;		(*Commande externe de marche de la source en automatique*)
	PRM_HV:				REAL;

	DEF_Source:			PRCDEF;

END_VAR


VAR_INPUT PERSISTENT
	(*Entité*)
	IsComponent:		BOOL;			(*entité : composant*)
	IdXML:				STRING;			(*nom entité : identifiant pour recherche dans dico*)
	TagXML:				UINT;			(*nom entité : identifiant pour recherche dans dico*)
	IdParent:			STRING;			(*MNEMO de l'appelant*)
	MNEMO:				STRING;			(*MNEMO de l'entité*)
END_VAR

VAR_OUTPUT
	OUT_ITLCK_EAU			AT%Q*:		BOOL;			(* sortie interlock eau*)
	OUT_ITLCK_VIDE			AT%Q*:		BOOL;			(* sortie interlock vide*)
	OUT_ITLCK_CHAMBRE		AT%Q*:		BOOL;			(* sortie interlock chambre*)
	OUT_ITCLK_EX			AT%Q*:		BOOL;			(* sortie interlock externe*)

	OUT_HV_ON				AT%Q*:		BOOL;			(* Marche Source*)
	OUT_HV_OFF				AT%Q*:		BOOL;			(* Arrêt Source*)

	AO_QHV:					ANALOG_OUTPUT;				(*sortie analogique alimentation HT*)
	OUT_QHV					AT%Q*:		INT;			(*Consigne Filament*)

	STATE_HV:			BOOL;							(*demande de mise en marche de la source en cours*)
	STATE_HV_ON:		BOOL;							(*Source en marche*)

	STATE_V_HV:			REAL;							(*HT appliqué*)
	STATE_I_FIL:		REAL;							(*Courant de filament*)

	STATE_POWER:		REAL;							(*Puissance appliquée en %*)

	STATE_NOK:			BOOL;							(*Alimentation en défaut*)
	STATE_READY:		BOOL;
END_VAR
VAR
	(*Gestion perte brève du retour IN_HVON*)
	TIMER_ON:			TP;
	FD_ON:				F_TRIG;
END_VAR

HV.IdParent := MNEMO;
HV.IdXML := '16';
HV.TagXML := 1;
HV.MNEMO := CONCAT(MNEMO,'_HV');

(*Défaut*)
HV.DEF_Off.IdXML				:=	'3';
HV.DEF_Off.TagXML				:=	3;
HV.DEF_On.IdXML					:=	'3';
HV.DEF_On.TagXML				:=	1;
HV.DEF_Off_Auto.IdXml			:=	'3';
HV.DEF_Off_Auto.TagXml			:=	10;
HV.DEF_On_imposs.IdXml			:=	'3';
HV.DEF_On_imposs.TagXml			:=	5;
HV.DEF_Off_imposs.IdXml			:=	'3';
HV.DEF_Off_imposs.TagXml		:=	8;

DEF_Source.IdXML				:=	'14';
DEF_Source.TagXML				:=	19;


AI_FIL(
	CONF_Max:= 1.0,		(*TODO Range*)
	CONF_Min:= 0.0,
	CONF_Bipolar:=FALSE ,
	CONF_Range:= 1,
	INPUT:= IN_FILQ );

AI_HV(
	CONF_Max:= 10.0,	(*TODO Range*)
	CONF_Min:= 0.0,
	CONF_Bipolar:=FALSE ,
	CONF_Range:= 1,
	INPUT:= IN_HVQ );



(*Temporisation HV.STATE_ON sur perte brève de IN_HVON *)
FD_ON.CLK := IN_HVON;
FD_ON();

TIMER_ON.IN := FD_ON.Q;
TIMER_ON.PT := T#20ms;
TIMER_ON();

HV(
	RESET:= RESET,
	MANUAL:= MANUAL,
	IN_ON := IN_HVON OR TIMER_ON.Q,
	CO_On:=CO_SRC ,
	EN_On_INT:=DOOR AND WATER AND VAC AND  (I_CR_OK OR (STATE_POWER = 0)),
	EN_Off_INT:= TRUE,
	CONF_Type_Actuator := 0,
	CONF_EN_On := 1,
	CONF_DI_Off:= FALSE,
	CONF_DI_On:= TRUE,
	CONF_No_Safety_Auto:=FALSE,
	CONF_Tim_Valid_On:= T#30s,
	CONF_Tim_Valid_Off:= T#2s,
	OUT_On=>,
	STATE_On=>STATE_HV_ON,
	STATE_Nok=> );

HV.DEF_Off.DELAY := T#20s;
HV.DEF_On.DELAY := T#60s;

(*Demande marche HT*)
OUT_HV_ON := HV.OUT_On;
STATE_HV := HV.OUT_On;

(*Demande arrêt HT*)
OUT_HV_OFF:= NOT HV.OUT_On;

(*Gestion de la sortie analogique filament*)
IF NOT STATE_HV_ON OR RESET THEN
	AO_QHV.Value := 0.0;
ELSIF MANUAL THEN
	AO_QHV.Value := PRM_POWER;
ELSE
	AO_QHV.Value := I_POWER;
END_IF;
AO_QHV(
	CONF_Max:=100,
	CONF_Min:= 0,
	CONF_Bipolar:=FALSE,
	CONF_Range:=1 );

OUT_QHV := AO_QHV.OUTPUT;

STATE_V_HV:= AI_HV.Value;
STATE_I_FIL:= AI_FIL.Value;
STATE_POWER := AO_QHV.Value;

(*gestion des interlock*)
OUT_ITLCK_EAU:= WATER;
OUT_ITLCK_VIDE:= VAC;
OUT_ITLCK_CHAMBRE:= DOOR;
OUT_ITCLK_EX:= DOOR;


(*Gestion des défauts*)
DEF_Source.CONDITION	:=	IN_ERROR;
DEF_Source.DELAY		:=	T#1s;
DEF_Source();

(*Retour Source en défaut*)
STATE_NOK:= HV.STATE_Nok OR DEF_Source.DEF;

STATE_READY:= WATER AND DOOR AND VAC AND I_CR_OK;

END_FUNCTION_BLOCK

// ---- POUs/Composant/EVAP/BLOCK_SWEEP_TELEMARK_PROG.TcPOU
FUNCTION_BLOCK BLOCK_SWEEP_TELEMARK_PROG

(* Gestion d'un controleur de balayage telemark programmable 16 motifs *)

(****************historique des versions*****************************)

(* Version 1-0 - GV - 01/15 - VERSION INIITIALE EVA760 n°12 - 8866 *)

(*************************************************************************)

VAR_INPUT
	MANUAL:					BOOL;		(*Mode de pilotage manuel *)
	RESET:					BOOL;		(*Condition de réiinitialisation de la fonction *)
	DOOR:					BOOL;		(*Interlock porte*)
	WATER:					BOOL;		(*Interlock eau*)

	DEF_Arret_Auto:			PRCDEF;	(* défaut d'arrêt automatique du balayage*)
	DEF_Marche_imposs:		PRCDEF;	(* défaut de marche du balayage non autorisée*)

	CO_On:					BOOL;		(*Demande de marche en mode automatique*)

	PRM_NbBal:				USINT:=1;	(*Commande de position*)
END_VAR

VAR
	TIMER_Valid_On:		TON;

	(* Variables demande en mode manuel*)
	M_RemLoc:			BOOL;	(* Ordre Remote/Local du module de balayage *)
	RCP_M_RemLoc:		BOOL;	(* Bit de reception de l'ordre Remote/Local du module de balayage *)
	VAR_RemLoc:			BOOL;	(* Variable intermédiare de l'ordre Remote/Local *)

	M_On:				BOOL;	(* Ordre Marche/Arrêt du module de balayage *)
	RCP_M_On:			BOOL;	(* Bit de reception de l'ordre de Marche/Arrêt du module de balayage *)
	VAR_On:				BOOL;	(* Variable intermédiaire de marche du module de balayage*)
END_VAR

VAR_OUTPUT
	(*variable d'état d'autorisation*)
	AUTOR_Rem_IHM:		BOOL;			(*indique que le mode Remote est autorisée en mode manuel depuis l'IHM*)
	AUTOR_Loc_IHM:		BOOL;			(*indique que le mode Local est autorisée en mode manuel depuis l'IHM*)
	AUTOR_On_IHM:		BOOL;			(*indique que la mise en marche du module est autorisée en mode manuel depuis l'IHM*)
	AUTOR_Off_IHM:		BOOL;			(*indique que l'arrêt du module est autorisée en mode manuel depuis l'IHM*)

	OUT_PSEL0:			BOOL;		(*sélection du motif*)
	OUT_PSEL1:			BOOL;		(*sélection du motif*)
	OUT_PSEL2:			BOOL;		(*sélection du motif*)
	OUT_PSEL3:			BOOL;		(*sélection du motif*)
	OUT_SWP_ON_OFF:		BOOL;		(*Marche/Arrêt balayage en mode Remote*)
	OUT_REM_LOC:		BOOL;		(*Mode Remote/Local*)
	STATE_NbBal:		USINT;
	STATE_BAL:			STRING;
	STATE_REM:			BOOL;		(*Module de balayage en mode Remote*)
	STATE_LOC:			BOOL;		(*Module de balayage en mode Local*)
	STATE_ON:			BOOL;		(*Module de balayage en marche*)
	STATE_OFF:			BOOL;		(*Module de balayage à l'arrêt*)
END_VAR


VAR_INPUT PERSISTENT

	PRM_BAL: 		ARRAY[0..16] OF STRING;		(*nom du programme de balayage*)

	(*Entité*)
	IsComponent:	BOOL;			(*entité : composant*)
	IdXML:			STRING;			(*nom entité : identifiant pour recherche dans dico*)
	TagXML:			UINT;			(*nom entité : identifiant pour recherche dans dico*)
	IdParent:		STRING;			(*MNEMO de l'appelant*)
	MNEMO:			STRING;			(*MNEMO de l'entité*)
END_VAR

DEF_Arret_Auto.IdXml			:=	'3';
DEF_Arret_Auto.TagXml			:=	10;

DEF_Marche_imposs.IdXml			:=	'3';
DEF_Marche_imposs.TagXml		:=	5;

(* Gestion des ordres en mode manuel *)
	RCP_M_RemLoc		:=	M_RemLoc;
	RCP_M_On			:=	M_On;

(*gestion des bits d'autorisation en mode manuel*)
	AUTOR_Rem_IHM		:=	NOT RESET AND NOT VAR_RemLoc  AND MANUAL;
	AUTOR_Loc_IHM		:=	NOT RESET  AND VAR_RemLoc  AND MANUAL;
	AUTOR_On_IHM		:=	NOT RESET AND NOT Var_On AND MANUAL AND DOOR AND WATER;
	AUTOR_Off_IHM		:=	NOT RESET AND VAR_On AND MANUAL;

(*défaut d'arrêt automatique du balyage *)
	DEF_Arret_Auto.CONDITION :=		(NOT DOOR
									OR  NOT WATER
									OR NOT VAR_RemLoc)
									AND VAR_On AND NOT RESET;
	DEF_arret_auto.DELAY:=T#0ms;
	DEF_Arret_Auto();

(* Défaut de marche du balayage non autorisée en automatique*)
	DEF_marche_imposs.CONDITION:=	NOT MANUAL AND CO_On AND (NOT DOOR OR NOT WATER)
									AND NOT RESET;
	DEF_marche_imposs.DELAY := T#0ms;
	DEF_marche_imposs();

(*gestion des variables intermédiare*)
(* Mode Local*)
	IF	RCP_M_RemLoc AND AUTOR_Loc_IHM OR RESET THEN
				Var_RemLoc 	:= 	FALSE;
(*Mode Remote*)
	ELSIF	NOT MANUAL OR ( RCP_M_RemLoc AND AUTOR_Rem_IHM) THEN
				Var_RemLoc 	:= 	TRUE;
	END_IF

(* Arrêt Balayage*)
	IF 		(NOT CO_On AND NOT MANUAL)
			OR ( RCP_M_On AND AUTOR_Off_IHM) OR DEF_arret_auto.DEF OR RESET
			THEN
				Var_On 				:= 	FALSE;
(*Marche Balayage*)
	ELSIF	( CO_On AND NOT MANUAL)
			 OR 	( RCP_M_On AND AUTOR_On_IHM) THEN
				Var_On 				:= 	TRUE;
	END_IF;

(*SORTIE Mode Remote/Local*)
	OUT_REM_LOC		:= 	VAR_RemLoc;
	OUT_SWP_ON_OFF	:=	VAR_On;

(*affectation des bits d'état*)
	STATE_REM			:=	OUT_REM_LOC;
	STATE_LOC			:=	NOT OUT_REM_LOC;
	STATE_OFF			:=	NOT OUT_SWP_ON_OFF;

(*indicateur  STATE_ON*)
TIMER_Valid_On.IN	:=	OUT_SWP_ON_OFF;
TIMER_Valid_On(PT:=T#500ms);
STATE_ON			:=	Timer_Valid_On.Q;


(*Selection du mode de balayage*)
CASE PRM_NbBal OF
		16:
			OUT_PSEL0 := TRUE;
			OUT_PSEL1 := TRUE;
			OUT_PSEL2 := TRUE;
			OUT_PSEL3 := TRUE;
		15:
			OUT_PSEL0 := FALSE;
			OUT_PSEL1 := TRUE;
			OUT_PSEL2 := TRUE;
			OUT_PSEL3 := TRUE;
		14:
			OUT_PSEL0 := TRUE;
			OUT_PSEL1 := FALSE;
			OUT_PSEL2 := TRUE;
			OUT_PSEL3 := TRUE;
		13:
			OUT_PSEL0 := FALSE;
			OUT_PSEL1 := FALSE;
			OUT_PSEL2 := TRUE;
			OUT_PSEL3 := TRUE;
		12:
			OUT_PSEL0 := TRUE;
			OUT_PSEL1 := TRUE;
			OUT_PSEL2 := FALSE;
			OUT_PSEL3 := TRUE;
		11:
			OUT_PSEL0 := FALSE;
			OUT_PSEL1 := TRUE;
			OUT_PSEL2 := FALSE;
			OUT_PSEL3 := TRUE;
		10:
			OUT_PSEL0 := TRUE;
			OUT_PSEL1 := FALSE;
			OUT_PSEL2 := FALSE;
			OUT_PSEL3 := TRUE;
		9:
			OUT_PSEL0 := FALSE;
			OUT_PSEL1 := FALSE;
			OUT_PSEL2 := FALSE;
			OUT_PSEL3 := TRUE;
		8:
			OUT_PSEL0 := TRUE;
			OUT_PSEL1 := TRUE;
			OUT_PSEL2 := TRUE;
			OUT_PSEL3 := FALSE;
		7:
			OUT_PSEL0 := FALSE;
			OUT_PSEL1 := TRUE;
			OUT_PSEL2 := TRUE;
			OUT_PSEL3 := FALSE;
		6:
			OUT_PSEL0 := TRUE;
			OUT_PSEL1 := FALSE;
			OUT_PSEL2 := TRUE;
			OUT_PSEL3 := FALSE;
		5:
			OUT_PSEL0 := FALSE;
			OUT_PSEL1 := FALSE;
			OUT_PSEL2 := TRUE;
			OUT_PSEL3 := FALSE;
		4:
			OUT_PSEL0 := TRUE;
			OUT_PSEL1 := TRUE;
			OUT_PSEL2 := FALSE;
			OUT_PSEL3 := FALSE;
		3:
			OUT_PSEL0 := FALSE;
			OUT_PSEL1 := TRUE;
			OUT_PSEL2 := FALSE;
			OUT_PSEL3 := FALSE;
		2:
			OUT_PSEL0 := TRUE;
			OUT_PSEL1 := FALSE;
			OUT_PSEL2 := FALSE;
			OUT_PSEL3 := FALSE;
		1:
			OUT_PSEL0 := FALSE;
			OUT_PSEL1 := FALSE;
			OUT_PSEL2 := FALSE;
			OUT_PSEL3 := FALSE;
END_CASE

STATE_NbBal := PRM_NbBal;

IF STATE_NbBal > 0 THEN
	STATE_BAL:= PRM_BAL[STATE_NbBal];
ELSE
	STATE_BAL:= '';
END_IF

(* Reset des ordres*)
	IF M_RemLoc AND RCP_M_RemLoc THEN
		M_RemLoc		:= FALSE;
	END_IF
	IF M_On	AND RCP_M_On THEN
		M_On			:=	FALSE;
	END_IF

END_FUNCTION_BLOCK

// ---- POUs/Composant/EVAP/BLOCK_TELEMARK_DIGITAL_SWEEP.TcPOU
FUNCTION_BLOCK BLOCK_TELEMARK_DIGITAL_SWEEP

(* Gestion d'un controleur de balayage telemark Digital Sweep 8 motifs*)

(****************historique des versions*****************************)

(* Version 1-0 - GV - 22/05/15 - VERSION INIITIALE EVA450 n°17 - 8950 *)
(* Version 2-0 - HG - 06/11/23 - Ajout sorties interlock et remote 14035
									Ajout Timer_valid_off*)

(*************************************************************************)

VAR_INPUT
	MANUAL:					BOOL;		(*Mode de pilotage manuel *)
	RESET:					BOOL;		(*Condition de réinitialisation de la fonction *)
	DOOR:					BOOL;		(*Porte fermée*)

	I_SW_REM:				BOOL;		(*Balayage en mode remote*)
	I_SW_RUN:				BOOL;		(*Balayage en marche*)
	I_SW_RDY:				BOOL;		(*Balayage prêt*)

	PRM_NbBal:				USINT:=1;	(*Commande de position*)
	
	CO_Remote:				BOOL;		(*Demande d'activation du mode remote en automatique*)
END_VAR

VAR
	TIMER_Valid_On:			TON;
	TIMER_Valid_Off:		TOF;
	M_Remote:				BOOL;	(* Ordre de changement commande remote *)
	RCP_M_Remote:			BOOL;	(* Bit de reception de l'ordre de remote du module de balayage*)
	VAR_Remote:				BOOL;	(* Variable intermédiaire commande remote du module de balayage*)
END_VAR

VAR_OUTPUT
	OUT_SWB1:			BOOL;		(*sélection du motif*)
	OUT_SWB2:			BOOL;		(*sélection du motif*)
	OUT_SWB3:			BOOL;		(*sélection du motif*)
	OUT_SWB4:			BOOL;		(*sélection du motif*)
	OUT_ITLK:			BOOL;		(*Interlock*)
	OUT_RMT:			BOOL;		(*Remote*)
	STATE_NbBal:		USINT;
	STATE_BAL:			STRING;
	STATE_REM:			BOOL;		(*Module de balayage en mode Remote*)
	STATE_LOC:			BOOL;		(*Module de balayage en mode Local*)
	STATE_ON:			BOOL;		(*Module de balayage en marche*)
	STATE_OFF:			BOOL;		(*Module de balayage à l'arrêt*)
	STATE_RDY:			BOOL;		(*Module de balayage à prêt*)
	AUTOR_Remote_IHM:			BOOL;		(*indique que le changement mode remote est autorisé en mode manuel depuis l'IHM*)
	AUTOR_Remote_PLC:			BOOL;		(*indique que le changement more remote est autorisé en mode automatique depuis l'automate*)
END_VAR


VAR_INPUT PERSISTENT

	PRM_BAL: 		ARRAY[0..8] OF STRING;		(*nom du programme de balayage*)

	(*Entité*)
	IsComponent:	BOOL;			(*entité : composant*)
	IdXML:			STRING;			(*nom entité : identifiant pour recherche dans dico*)
	TagXML:			UINT;			(*nom entité : identifiant pour recherche dans dico*)
	IdParent:		STRING;			(*MNEMO de l'appelant*)
	MNEMO:			STRING;			(*MNEMO de l'entité*)
END_VAR

(* Gestion des ordres en mode manuel *)
RCP_M_Remote			:=	M_Remote;

(*affectation des bits d'état*)
STATE_REM			:=	I_SW_REM;
STATE_LOC			:=	NOT I_SW_REM;
STATE_OFF			:=	NOT I_SW_RUN;
STATE_RDY			:=	I_SW_RDY;

(*indicateur  STATE_ON*)
TIMER_Valid_On.IN	:=	I_SW_RUN;
TIMER_Valid_On(PT:=T#500ms);
TIMER_Valid_Off.IN	:=	I_SW_RUN;
TIMER_Valid_Off(PT:=T#200ms);
STATE_ON			:=	Timer_Valid_On.Q AND TIMER_Valid_Off.Q;

(*gestion des bits d'autorisation en mode manuel*)
AUTOR_Remote_IHM		:=	NOT RESET AND MANUAL;
AUTOR_Remote_PLC		:=	NOT RESET AND NOT MANUAL;

(*Selection du mode de balayage*)
CASE PRM_NbBal OF
		8:
			OUT_SWB1 := FALSE;
			OUT_SWB2 := FALSE;
			OUT_SWB3 := FALSE;
			OUT_SWB4 := TRUE;
		7:
			OUT_SWB1 := TRUE;
			OUT_SWB2 := TRUE;
			OUT_SWB3 := TRUE;
			OUT_SWB4 := FALSE;
		6:
			OUT_SWB1 := FALSE;
			OUT_SWB2 := TRUE;
			OUT_SWB3 := TRUE;
			OUT_SWB4 := FALSE;
		5:
			OUT_SWB1 := TRUE;
			OUT_SWB2 := FALSE;
			OUT_SWB3 := TRUE;
			OUT_SWB4 := FALSE;
		4:
			OUT_SWB1 := FALSE;
			OUT_SWB2 := FALSE;
			OUT_SWB3 := TRUE;
			OUT_SWB4 := FALSE;
		3:
			OUT_SWB1 := TRUE;
			OUT_SWB2 := TRUE;
			OUT_SWB3 := FALSE;
			OUT_SWB4 := FALSE;
		2:
			OUT_SWB1 := FALSE;
			OUT_SWB2 := TRUE;
			OUT_SWB3 := FALSE;
			OUT_SWB4 := FALSE;
		1:
			OUT_SWB1 := TRUE;
			OUT_SWB2 := FALSE;
			OUT_SWB3 := FALSE;
			OUT_SWB4 := FALSE;
END_CASE
STATE_NbBal := PRM_NbBal;
IF STATE_NbBal > 0 THEN
	STATE_BAL:= PRM_BAL[STATE_NbBal];
ELSE
	STATE_BAL:= '';
END_IF

(*gestion interlock*)
OUT_ITLK	:=	NOT RESET AND DOOR;

(*gestion remote*)
IF	(CO_Remote AND AUTOR_Remote_PLC)
		 OR 	(RCP_M_Remote AND NOT VAR_Remote AND AUTOR_Remote_IHM) THEN
			VAR_Remote 		:= 	TRUE;
ELSIF (NOT CO_Remote AND NOT RESET AND NOT MANUAL)
		OR 	(RCP_M_Remote AND VAR_Remote AND AUTOR_Remote_IHM)
		OR 	RESET THEN
			VAR_Remote		:=	FALSE;
END_IF;
OUT_RMT	:=	VAR_Remote;

(* Reset des ordres*)
IF M_Remote	AND RCP_M_Remote THEN
	M_Remote			:=	FALSE;
END_IF

END_FUNCTION_BLOCK

// ---- POUs/Composant/EVAP/BLOCK_XTAL.TcPOU
FUNCTION_BLOCK BLOCK_XTAL
VAR_INPUT
	I_APPLY_PARAMETER:		BOOL;

	RESET:					BOOL;
	MANUAL:					BOOL;
	CO_OUV_CACHE:			BOOL;		(*Demande d'ouverture du cache*)

	IN_QF:					BOOL;		(*Quartz en panne*)
	IN_RATE:				REAL;		(*Vitesse de dépot mesurée sur le quartz*)
	IN_FREQ:				REAL;		(*Frequence du quartz*)
	IN_THICKNESS:			REAL;		(*Epaisseur*)
	IN_LIFE:				REAL;		(*Vie du quartz*)
	IN_ACTIVITY:			REAL;		(*Activité du quartz*)
	IN_ACTIVE_CRYSTAL:		USINT;		(*Numéro du crystal active*)

	(*Consigne*)
	CONS_MATERIAL:	 		STRING;		(*Materiau*)
	CONS_POID:				REAL;		(*Poids du quartz pour la calcul du quartz*)
	CONS_ZRATIO:			REAL;		(*Valeur du Zratio*)
	CONS_DENSITE:			REAL;		(*Valeur de densité*)
	CONS_TOOLING:			REAL;		(*Facteur de correction de chaque quartz*)

(*Défauts*)
	DEF_QZ:					PRCDEF;	(*Défaut quartz*)

(*Alarme*)
	ALM_SURV_ACTIVITY:		PRCDEF;		(*Alarme surveillance activité quartz*)
	ALM_SURV_LIFE:			PRCDEF;		(*Alarme surveillance vie quartz*)
(*Evenements*)
	EV_SWITCH_XTAL:			PRCDEF;		(*Evenement en cas de basculement sur le quartz principal*)
	EV_SWITCH_BACKUP:		PRCDEF;		(*Evenement en cas de basculement sur le quartz de secours*)

(*Opérations*)
	CQZ:					BLOCK_ACTUATOR2;

END_VAR

VAR_OUTPUT
	STATE_LIFE:				REAL;
	STATE_ACTIVITY:			REAL;
	STATE_FREQUENCY:		REAL;
	STATE_THICKNESS:		REAL;
	STATE_RATE:				REAL;
	STATE_MATERIAL:			STRING;
	STATE_NOK:				BOOL;
	OUT_MATERIAL:			STRING;
	OUT_POIDS:				REAL;
	OUT_ZRATIO:				REAL;
	OUT_DENSITE:			REAL;
	OUT_TOOLING:			REAL;

	OUT_CQZ AT%Q*:			BOOL;		(*Ouverture du cache Quartz *)


END_VAR


VAR_INPUT PERSISTENT
	(*Entité*)
	IsComponent:	BOOL;			(*entité : composant*)
	IdXML:			STRING;			(*nom entité : identifiant pour recherche dans dico*)
	TagXML:			UINT;			(*nom entité : identifiant pour recherche dans dico*)
	IdParent:		STRING;			(*MNEMO de l'appelant*)
	MNEMO:			STRING;			(*MNEMO de l'entité*)

	PRM_Seuil_Life:			REAL;	(*Seuil d'alarme pour la vie du quartz*)
	PRM_Seuil_Activity:		REAL;	(*Seuil d'alarme pour l'activité du quartz*)
END_VAR

VAR
END_VAR

TagXML:= 9;
IdXML:=	'16';
DEF_QZ.IdXML := '14';
DEF_QZ.TagXML := 3;

CQZ.IdParent:= MNEMO;
CQZ.IdXML := '4';
CQZ.TagXML := 1;

(*Défaut*)
CQZ.DEF_Off_Auto.IdXml		:=	'3';
CQZ.DEF_Off_Auto.TagXml		:=	10;
CQZ.DEF_On_imposs.IdXml		:=	'3';
CQZ.DEF_On_imposs.TagXml	:=	5;
CQZ.DEF_Off_imposs.IdXml	:=	'3';
CQZ.DEF_Off_imposs.TagXml	:=	8;

(*Alarme surveillance*)
ALM_SURV_ACTIVITY.IdXml		:=	'0';
ALM_SURV_ACTIVITY.TagXml	:=	8;
ALM_SURV_ACTIVITY.Groupe	:=	1;

ALM_SURV_LIFE.IdXML			:=	'0';
ALM_SURV_LIFE.TagXML		:=	8;
ALM_SURV_LIFE.Groupe		:= 	1;

EV_SWITCH_XTAL.IdXML		:=	'14';
EV_SWITCH_XTAL.TagXML		:=	23;
EV_SWITCH_XTAL.Groupe		:=	3;

EV_SWITCH_BACKUP.IdXML		:=	'14';
EV_SWITCH_BACKUP.TagXML		:=	22;
EV_SWITCH_BACKUP.Groupe		:= 	3;

IF I_APPLY_PARAMETER THEN
	OUT_DENSITE 	:=	CONS_DENSITE;
	OUT_POIDS		:=	CONS_POID;
	OUT_ZRATIO		:=	CONS_ZRATIO;
	OUT_MATERIAL	:= 	CONS_MATERIAL;
	OUT_TOOLING		:=	CONS_TOOLING;
END_IF

CQZ(
	RESET:= RESET,
	MANUAL:= MANUAL,
	CO_On:=CO_OUV_CACHE ,
	EN_On_INT:=TRUE,
	EN_Off_INT:= TRUE,
	CONF_No_Safety_Auto:=FALSE ,
	CONF_EN_On:= 0 ,
	CONF_Tim_Valid_On:= T#0ms,
	CONF_Tim_Valid_Off:= T#0ms
);

OUT_CQZ:= CQZ.OUT_On;


STATE_FREQUENCY	:= 	IN_FREQ;
STATE_RATE		:= 	IN_RATE;
STATE_THICKNESS	:= 	IN_THICKNESS;
STATE_LIFE			:=	IN_LIFE;
STATE_ACTIVITY	:= 	IN_ACTIVITY;
STATE_MATERIAL	:=	OUT_MATERIAL;
STATE_NOK			:=	DEF_QZ.DEF;

(*Alarme Activité < Seuil d'activité limite*)
ALM_SURV_ACTIVITY.CONDITION	:=	(IN_ACTIVITY < PRM_Seuil_Activity);
ALM_SURV_ACTIVITY();

(*Alarme Vie > Seuil de vie limite*)
ALM_SURV_LIFE.CONDITION	:=	(IN_LIFE > PRM_Seuil_Life);
ALM_SURV_LIFE();

(*Evenement en cas de basculement sur le quartz principal*)
EV_SWITCH_XTAL.CONDITION		:=	CQZ.STATE_Off;
EV_SWITCH_XTAL();

(*Evenement en cas de basculement sur le quartz de secours*)
EV_SWITCH_BACKUP.CONDITION	:=	CQZ.STATE_On;
EV_SWITCH_BACKUP();


DEF_QZ(
		CONDITION:=	IN_QF,
		DELAY:=			T#0s);

END_FUNCTION_BLOCK

// ---- POUs/Composant/GAZ/BLOCK_MFC_ANA2.TcPOU
FUNCTION_BLOCK BLOCK_MFC_ANA2
(* Gestion débitmètre massique analogique*)

(****************historique des versions*****************************)

(* Version 1-0 - HG - VERSION INITIALE*)
(*Version 1-1 - AB - interface standard et ajout entrée désactivation surveillance - affaire 7018*)

(*************************************************************************)

VAR_INPUT
(*informations générales*)
	RESET:					BOOL;		(* Condition de réinitialisation de la fonction *)
	PRM_Flow:				REAL;		(* ~ (OPC : 1 : available for OPC-clients) *)	(* Consigne débit gaz*)

	DEF_SURV:				PRCDEF;	(* ~ (OPC : 1 : available for OPC-clients) *)	(* Défaut surveillance débit*)
	ALM_SURV:				PRCDEF;	(* ~ (OPC : 1 : available for OPC-clients) *)	(* Alarme surveillance débit*)
	VAR_DEF_SURV:			SURVPRC;	(* ~ (OPC : 1 : available for OPC-clients) *)	(* Condition defaut surveillance débit*)
	VAR_ALM_SURV:			SURVPRC;	(* ~ (OPC : 1 : available for OPC-clients) *)	(* Condition alarme surveillance débit*)

	I_SURV_DISABLE:			BOOL;		(* I_STANDARD -- option de desactivation de la surveillance du débit venant du bloc ligne de gaz*)

	IN_Measure:				ANALOG_INPUT;									(* entrée analogique débit*)
END_VAR

VAR_OUTPUT
	STATE_Flow:				REAL;		(* ~ (OPC : 1 : available for OPC-clients) *)	(* Débit gaz appliqué*)
	CONF_Util_Max_Flow:		REAL:=1;		(* ~ (OPC : 1 : available for OPC-clients) *)	(* Débit max gaz utilisé*)
	STATE_NOK:				BOOL;		(* ~ (OPC : 1 : available for OPC-clients) *)	(* Débitmètre en défaut*)

	OUT_SetPoint:			ANALOG_OUTPUT;								(* Sortie analogique débit gaz*)
END_VAR

VAR_INPUT PERSISTENT
(*Configuration*)
	CONF_Nom_Max_Flow:		REAL:=1;		(* ~ (OPC : 1 : available for OPC-clients) *)	(* Débit max gaz nominal débitmètre*)
	CONF_Nom_Coef:			REAL:=1;		(* ~ (OPC : 1 : available for OPC-clients) *)	(* Coefficient gaz nominal débitmètre*)
	CONF_Util_Coef:			REAL:=1;		(* ~ (OPC : 1 : available for OPC-clients) *)	(* Coefficient gaz utilisé*)
	CONF_Nom_Name:			STRING;		(*Nom du gaz nominal*)
	CONF_Util_Name:			STRING;		(*Nom du gaz utilisé*)

	(*Entité*)
	IsComponent:		BOOL;			(*entité : composant*)
	IdXML:				STRING;			(*nom entité : identifiant pour recherche dans dico*)
	TagXML:				UINT;			(*nom entité : identifiant pour recherche dans dico*)
	IdParent:			STRING;			(*MNEMO de l'appelant*)
	MNEMO:				STRING;			(*MNEMO de l'entité*)
END_VAR

VAR

END_VAR

IdXML					:=	'7';
TagXML					:=	1;

DEF_SURV.IdXml			:=	'0';
DEF_SURV.TagXml			:=	7;

ALM_SURV.IdXml			:=	'0';
ALM_SURV.TagXml			:=	8;
ALM_SURV.Groupe			:=	1;

(*Débit max utile*)
IF CONF_Nom_Coef > 0.0 THEN
	CONF_Util_Max_Flow	:=	CONF_Nom_Max_Flow * CONF_Util_Coef / CONF_Nom_Coef;
ELSE
	CONF_Util_Max_Flow	:=	0.0;
END_IF;

(*Traitement de l'entrée analogique*)
IN_Measure(
	CONF_Range:=0.5,					(*si 0-10V*)
	CONF_Max:=CONF_Util_Max_Flow,
	CONF_Min:=0.0,
	CONF_Bipolar:=FALSE);

(*Retour débit*)
IF CONF_Nom_Coef > 0.0 THEN
	STATE_Flow		:=	IN_Measure.Value * CONF_Util_Coef / CONF_Nom_Coef;
ELSE
	STATE_Flow		:=	0.0;
END_IF

(*Consigne débit*)
IF NOT reset AND PRM_Flow>0.0 AND CONF_Util_Coef > 0.0 THEN
	OUT_SetPoint.Value :=	PRM_Flow * CONF_Nom_Coef / CONF_Util_Coef;
ELSE
	OUT_SetPoint.Value	:=	0.0;
END_IF;

STATE_NOK		:=	alm_surv.DEF OR def_surv.DEF;

(*Traitement de la sortie analogique*)
OUT_SetPoint(
	CONF_Range := 0.5,        (*si 0..10V*)
	CONF_Max:=CONF_Util_Max_Flow ,
	CONF_Min:=0 ,
	CONF_Bipolar:=FALSE);
	

(*desactivation de la surveillance*)
ALM_SURV.DISABLE	:=	I_SURV_DISABLE;
DEF_SURV.DISABLE	:=	I_SURV_DISABLE;


(*Défaut surveillance*)
VAR_ALM_SURV(MEASURE:=STATE_Flow , SETPOINT:= PRM_Flow);
ALM_SURV.CONDITION	:=	VAR_ALM_SURV.CONDITION ;
ALM_SURV();

VAR_DEF_SURV(MEASURE:=STATE_Flow , SETPOINT:= PRM_Flow);
DEF_SURV.CONDITION	:=	VAR_DEF_SURV.CONDITION ;
DEF_SURV();

END_FUNCTION_BLOCK

// ---- POUs/Composant/GAZ/BLOCK_MFC_BKH.TcPOU
FUNCTION_BLOCK BLOCK_MFC_BKH
(* Gestion débitmètre massique Bronkhorst*)

(****************historique des versions*****************************)

(* Version 1-0 - HG - VERSION INITIALE*)
(*Version 1-1 - AB - interface standard et ajout entrée désactivation surveillance - affaire 6970*)
(*Version 2-0 - HG - Adaptation pour journal des évènements externe - 27/06/2011*)

(*************************************************************************)

VAR_INPUT
(*informations générales*)
	RESET:					BOOL;		(* Condition de réinitialisation de la fonction *)
	PRM_Flow:				REAL;		(* ~ (OPC : 1 : available for OPC-clients) *)	(* Consigne débit gaz*)

	DEF_SURV:				PRCDEF;	(* ~ (OPC : 1 : available for OPC-clients) *)	(* Défaut surveillance débit*)
	ALM_SURV:				PRCDEF;	(* ~ (OPC : 1 : available for OPC-clients) *)	(* Alarme surveillance débit*)
	VAR_DEF_SURV:			SURVPRC;	(* ~ (OPC : 1 : available for OPC-clients) *)	(* Condition defaut surveillance débit*)
	VAR_ALM_SURV:			SURVPRC;	(* ~ (OPC : 1 : available for OPC-clients) *)	(* Condition alarme surveillance débit*)

	I_SURV_DISABLE:			BOOL;		(* I_STANDARD -- option de desactivation de la surveillance du débit venant du bloc ligne de gaz*)
END_VAR

VAR_OUTPUT
	STATE_Flow:				REAL;		(* ~ (OPC : 1 : available for OPC-clients) *)	(* Débit gaz appliqué*)
	CONF_Util_Max_Flow:		REAL:=1;		(* ~ (OPC : 1 : available for OPC-clients) *)	(* Débit max gaz utilisé*)
	STATE_Com:				BOOL;		(* ~ (OPC : 1 : available for OPC-clients) *)	(* Etat communication profibus*)
	STATE_NOK:				BOOL;		(* ~ (OPC : 1 : available for OPC-clients) *)	(* Débitmètre en défaut*)
END_VAR

VAR_INPUT PERSISTENT
(*Configuration*)
	CONF_Nom_Max_Flow:	REAL:=1;		(* ~ (OPC : 1 : available for OPC-clients) *)	(* Débit max gaz nominal débitmètre*)
	CONF_Nom_Coef:		REAL:=1;		(* ~ (OPC : 1 : available for OPC-clients) *)	(* Coefficient gaz nominal débitmètre*)
	CONF_Util_Coef:		REAL:=1;		(* ~ (OPC : 1 : available for OPC-clients) *)	(* Coefficient gaz utilisé*)
	CONF_Nom_Name:		STRING;		(*Nom du gaz nominal*)
	CONF_Util_Name:		STRING;		(*Nom du gaz utilisé*)

	(*Entité*)
	IsComponent:		BOOL;			(*entité : composant*)
	IdXML:				STRING;			(*nom entité : identifiant pour recherche dans dico*)
	TagXML:				UINT;			(*nom entité : identifiant pour recherche dans dico*)
	IdParent:			STRING;			(*MNEMO de l'appelant*)
	MNEMO:				STRING;			(*MNEMO de l'entité*)
END_VAR

VAR
	OUT_Setpoint	AT %Q*:	ARRAY[0..1] OF USINT;	(* Sortie consigne débit*)
	IN_Measure		AT %I*:	ARRAY[0..1] OF USINT;	(* Retour mesure débit*)
	IN_Status		AT %I*:	USINT;		(* Retour état communication*)
	VAR_Ret_flow:			REAL;
	VAR_Cons_flow:			REAL;
	VAR_Coef:				REAL;
	VAR_DW_Calcul:			DWORD;
	VAR_Comm_err:			BOOL;
	VAR_Process_err:		BOOL;
	VAR_Param_err:			BOOL;
	VAR_Type_err:			BOOL;
	VAR_Value_err:			BOOL;
	VAR_Cmd_err:			BOOL;
END_VAR

IdXML					:=	'7';
TagXML					:=	1;

DEF_SURV.IdXml			:=	'0';
DEF_SURV.TagXml			:=	7;

ALM_SURV.IdXml			:=	'0';
ALM_SURV.TagXml			:=	8;
ALM_SURV.Groupe			:=	1;

(*Débit max utile*)
IF CONF_Nom_Coef > 0.0 THEN
	CONF_Util_Max_Flow	:=	CONF_Nom_Max_Flow * CONF_Util_Coef / CONF_Nom_Coef;
ELSE
	CONF_Util_Max_Flow	:=	0.0;
END_IF;

(*Retour débit*)
IF CONF_Nom_Coef > 0.0 THEN
	VAR_Ret_Flow	:=	UINT_TO_REAL(IN_MEASURE[0]*16#FF+IN_MEASURE[1]);
	VAR_Ret_Flow	:=	(VAR_Ret_Flow*Conf_Nom_Max_Flow)/32000;
	STATE_Flow		:=	VAR_Ret_Flow * CONF_Util_Coef / CONF_Nom_Coef;
ELSE
	STATE_Flow		:=	0.0;
END_IF

(*Consigne débit*)
IF NOT reset AND PRM_Flow>0.0 AND CONF_Util_Coef > 0.0 THEN
	VAR_Cons_Flow	:=	PRM_Flow * CONF_Nom_Coef / CONF_Util_Coef;
ELSE
	VAR_Cons_Flow	:=	0.0;
END_IF;

IF CONF_Nom_Max_Flow>0 THEN
	VAR_DW_Calcul	:=	REAL_TO_DWORD((VAR_Cons_Flow*32000)/Conf_Nom_Max_Flow);
ELSE
	VAR_DW_Calcul	:=	REAL_TO_DWORD(0);
END_IF

OUT_Setpoint[1]	:=	DWORD_TO_USINT(VAR_DW_Calcul AND 16#FF);
OUT_Setpoint[0]	:=	DWORD_TO_USINT((VAR_DW_Calcul AND 16#FF00)/16#FF);

(*Retour état*)
VAR_Comm_err	:=	IN_Status.0;
VAR_Process_err	:=	IN_Status.1;
VAR_Param_err	:=	IN_Status.2;
VAR_Type_err	:=	IN_Status.3;
VAR_Value_err	:=	IN_Status.4;
VAR_Cmd_err	:=	IN_Status.5;
STATE_COM		:=	NOT VAR_comm_err AND NOT VAR_process_err AND NOT VAR_Param_err
					AND NOT VAR_type_err AND NOT VAR_value_err AND NOT VAR_Cmd_err;
STATE_NOK		:=	NOT state_com OR alm_surv.DEF OR def_surv.DEF;

(*desactivation de la surveillance*)
ALM_SURV.DISABLE	:=	I_SURV_DISABLE;
DEF_SURV.DISABLE	:=	I_SURV_DISABLE;

(*Défaut surveillance*)
VAR_ALM_SURV(MEASURE:=STATE_Flow , SETPOINT:= PRM_Flow);
ALM_SURV.CONDITION	:=	VAR_ALM_SURV.CONDITION ;
ALM_SURV();

VAR_DEF_SURV(MEASURE:=STATE_Flow , SETPOINT:= PRM_Flow);
DEF_SURV.CONDITION	:=	VAR_DEF_SURV.CONDITION ;
DEF_SURV();

END_FUNCTION_BLOCK

// ---- POUs/Composant/GAZ/BLOCK_MFC_BROOKS_NoCoE.TcPOU
FUNCTION_BLOCK BLOCK_MFC_BROOKS_NoCoE
(* Gestion débitmètre massique Brooks sur Ethercat*)

